IF stagingFunnel.enable THEN
stagingFunnel(
	openingDelay := HMIData.stagingFunnelOpenDelay, 
	openingDwell := HMIData.stagingFunnelOpeningTime,
	closingDwell := HMIData.stagingFunnelClosingTime,
	iOpened := iStagingFunnelOpened, 
	iClosed := iStagingFunnelClosed,  
	oClose => oStagingFunnelCloseOrPerfBreakerDown, 
	oOpen => oStagingFunnelOpenOrPerfBreakerUp
);
END_IF
	 
CASE HMIData.funnelFactorySelection OF
	FunnelSelection.NotInstalled:
		// Disable both funnels
		funnel.enable := FALSE;
		stagingFunnel.enable := FALSE;
		
	FunnelSelection.FunnelWithSensors:
		//
		funnel.enable := HMIData.funnelInUse;
		funnel.feedback := eActuatorFeedbackType.Both;
		stagingFunnel.enable := FALSE;
	
	FunnelSelection.FunnelWithoutSensors:
		//
		funnel.enable := HMIData.funnelInUse;
		funnel.feedback := eActuatorFeedbackType.None;
		stagingFunnel.enable := FALSE;
		
	FunnelSelection.TwoStageFunnelWithSensors:

		_fillerDroppingProductONS(CLK := filler.droppingProduct);
		IF _fillerDroppingProductONS.OSR THEN
			stagingFunnel.Open();
		ELSIF _fillerDroppingProductONS.OSF THEN
			stagingFunnel.Close();
		END_IF

		//
		funnel.enable := HMIData.funnelInUse;
		funnel.feedback := eActuatorFeedbackType.Both;
		stagingFunnel.enable := HMIData.funnelInUse;
		stagingFunnel.feedback := eActuatorFeedbackType.Both;
			 
	FunnelSelection.BagLoadingTray:
		funnel.enable := HMIData.funnelInUse;
		funnel.feedback := eActuatorFeedbackType.Both;
		stagingFunnel.enable := FALSE;
			 
END_CASE

//
sealBarTempSensor(
	busNodeOK := murrIOBusNode.ok,
	ptrTemperatureBytes := ADR(iHeaterBarTempInputs)
);
	 
//
IF sealBarTempSensor.reconfigureIO THEN
	murrIOBusNode.restartBusnodePulse.Trigger();		 
END_IF

//	 
sealBarHeater(
	enable := NOT safePowerFailure.active,
	temperatureSensor := sealBarTempSensor,
	temperatureSetpoint := TO_REAL(HMIData.sealBarTemperatureSetting),
	heaterPulse => 	oHeaterPulse,
	currentTemp => HMIData.sealBarTemperature
);	  

{region "timers"}
// Timers
sealTimer();
bagOpenFingerDelay();
vacuumHoldTimer(PT := TO_TIME(HMIData.vacuumDwell * 1000));
bagOpenCheckDelay();
bagDropTimer(PT := TO_TIME((HMIData.loadPlateDelay * 1000) + (HMIData.bagDropTime * 1000)));
{endregion}
		  
// Setup of HPA and load plate.  Use .Trigger() to run.
HPA.DwellSetting := TO_UINT(HMIData.hpaDwell * 1000);
HPA(Q => oHPAOn);
hpaServiceOnONS(CLK := HMIData.hpaserviceOn);

triggerLPAWhileFeedingONS(CLK := state.sb.releaseFeed = RELEASE_FEED_STATES.MovingJawOutAndFeedingBag);
IF HMIData.lpaDuringBagFeedEnable AND triggerLPAWhileFeedingONS.OSR THEN
	LPA.DwellSetting := TO_DINT(((bagDelivery.remainingLength - HMIData.bagSkirtLength) / TO_REAL(HMIData.bagForwardSpeed)) * 1000.0);
	LPA.Trigger();
END_IF
LPA(Q => oLPAOn);
	 
CASE HMIData.independentBagDeflatorSelection OF
	BagDeflatorSelection.NotInstalled:					// Disable IBD
		 													enableIBDDeflate := FALSE;
															enableIBDEject := FALSE;
	
	BagDeflatorSelection.IBDStandard:	// Enable IBD
															IF HMIData.IBDDeflateDwellTime <> 0 THEN
																enableIBDDeflate := TRUE;
															ELSE
																enableIBDDeflate := FALSE;
															END_IF
															
															IF HMIData.IBDPackageEjectAssistDwellTime <> 0 THEN
																enableIBDEject := TRUE;
															ELSE
																enableIBDEject := FALSE;
															END_IF
	 														
																 
	BagDeflatorSelection.IBDWithHingedPlate:	// Enable IBD with Hinged Plate
															
																 
	BagDeflatorSelection.MotorizedIBD:			// Enable motorized IBD
															IF HMIData.IBDDeflateDwellTime <> 0 THEN
																enableIBDDeflate := TRUE;
															ELSE
																enableIBDDeflate := FALSE;
															END_IF
															
															IF HMIData.IBDPackageEjectAssistDwellTime <> 0 THEN
																enableIBDEject := TRUE;
															ELSE
																enableIBDEject := FALSE;
															END_IF
END_CASE
		
(*  
CASE HMIData.bofSelection OF
	BagOpenFingersSelection.NotInstalled:					// Disable Bag Open
		 													enableBagOpen := FALSE;
															
	
	BagOpenFingersSelection.PneumaticWithBagOpenSensors:	// Enable Bag Open
															enableBagOpen := TRUE;
	
END_CASE
	 *)
		  enableBagOpen := HMIData.bagOpenEnable;

CASE HMIData.cycleStartButtonSelection OF
	PalmButtonSelection.NotInstalled:					// Dont' allow input to start bagger cycle
		 												startCycleReqFromPalmButtons := FALSE;
		 
	PalmButtonSelection.SinglePalmButton:				// Start using one side only
		 												startCycleReqFromPalmButtons := iRightPalmButton;
														
														// Trigger fault if left palm button is seen - should be set up for dual!	 
														IF iLeftPalmButton THEN
															palmButtonConfigError.Trigger();		 
														END_IF
		 
	PalmButtonSelection.DualPalmButton:					// Both buttons must be pressed
		 												startCycleReqFromPalmButtons := iRightPalmButton AND iLeftPalmButton;
															 
	PalmButtonSelection.LightedPalmButton:				
		// Lighted Murr palm button input comes from IO Link
		startCycleReqFromPalmButtons := iMurrTouchButtonOneStatus.0 OR iMurrTouchButtonTwoStatus.0;
		basicLightedPalmButton(
			baggerReady:= readyToRun AND NOT HMIData.sealBarNotAtTemperature.active, 
			baggerFaulted:= HMIData.faultActive, 
			baggerInCycle:= HMIData.inCycle, 
		);
		oMurrTouchbuttonOneState := oMurrTouchButtonTwoState := basicLightedPalmButton.IOLinkStateOutput;													 
														
    PalmButtonSelection.LightedPalmButtonAdvanced, PalmButtonSelection.DualLightedPalmButtonAdvanced:		
		// Lighted Murr palm button input comes from IO Link
		startCycleReqFromPalmButtons := iMurrTouchButtonOneStatus.0 OR iMurrTouchButtonTwoStatus.0;														 
		advancedLightedPalmButtonOne(
			IOLinkData := ADR(oMurrTouchButtonOneIOLinkOutputs),
			baggerReady := readyToRun 
							AND (NOT HMIData.sealBarNotAtTemperature.active) 
							AND (NOT HMIData.stopMachine) ,
			baggerFaulted := HMIData.faultActive,
			baggerInCycle := HMIData.inCycle,
			baggerExternalInhibited := printAndApply.state = PRINT_AND_APPLY_STATES.Inhibited,
			baggerHeatingUp := HMIData.sealBarNotAtTemperature.active AND sealBarHeater.heating,
			baggerCoolingDown := HMIData.sealBarNotAtTemperature.active AND sealBarHeater.cooling AND sealBarHeater.enable
		);	
        IF HMIData.cycleStartButtonSelection = PalmButtonSelection.DualLightedPalmButtonAdvanced THEN
			advancedLightedPalmButtonTwo(
				IOLinkData := ADR(oMurrTouchButtonTwoIOLinkOutputs),
				baggerReady := readyToRun 
							AND (NOT HMIData.sealBarNotAtTemperature.active) 
							AND (NOT HMIData.stopMachine) ,
				baggerFaulted := HMIData.faultActive,
				baggerInCycle := HMIData.inCycle,
				baggerExternalInhibited := printAndApply.state = PRINT_AND_APPLY_STATES.Inhibited,
				baggerHeatingUp := HMIData.sealBarNotAtTemperature.active AND sealBarHeater.heating,
				baggerCoolingDown := HMIData.sealBarNotAtTemperature.active AND sealBarHeater.cooling AND sealBarHeater.enable
			);	
		END_IF					  									 
END_CASE
startCycleReqFromPalmButtonsONS(CLK := startCycleReqFromPalmButtons);	 

// Stack Light active only if no 2nd palm button selected - they use the same IOLink port
IF HMIData.cycleStartButtonSelection <> PalmButtonSelection.DualLightedPalmButtonAdvanced THEN
	stackLight(
		IOLinkData:= ADR(oMurrStackLightOutputs), 
		baggerReady := readyToRun AND NOT HMIData.sealBarNotAtTemperature.active AND NOT HMIData.faultActive ,
		baggerFaulted := HMIData.faultActive,
		baggerInCycle := HMIData.inCycle,
		baggerExternalInhibited := printAndApply.state = PRINT_AND_APPLY_STATES.Inhibited ,
		bagsLow:= HMIData.bagLevelLow.active, 
		bagOpenRetryActive:= bagOpenRetryCount <> 0,
		baggerHeatingUp := HMIData.sealBarNotAtTemperature.active AND sealBarHeater.heating
	);	 
END_IF

		 
_auxIOPhysical(
	state := state,
	configIn1 := iAuxConfigInput1, 
	configIn2 := iAuxConfigInput2,
	bagsLow := HMIData.bagLevelLow.active,
	faultActive := HMIData.faultActive,
	inhibitCycle := printAndApply.inhibitCycle,
	printerDataReady := printerDataReady,
	waitingForFiller := filler.waitingForFiller,
	runExitConveyor := oRunExternalExitConveyor,
	fillerType := HMIData.fillerFactorySelection,
	factorySelection := HMIData.auxIOConfig,
	baggerOK => oAuxBaggerOk,
	readyForFiller => oAuxReadyForFiller,
	inhibitBagger => ,
	configOut1 => oAuxConfigOut1,
	configOut2 => oAuxConfigOut2,
);
	 
		  
_auxIORemote(
	state := state,	
	bagsLow := HMIData.bagLevelLow.active,
	faultActive := HMIData.faultActive,
	inhibitCycle := printAndApply.inhibitCycle,
	printerDataReady := printerDataReady,
	waitingForFiller := filler.waitingForFiller,
	runExitConveyor := oRunExternalExitConveyor,	
	activeFaults := GlobalObjects.CollectionOfActiveFaults.ObjNames,
	inhibitBagger => 
);

HMIData.baggerInhibited.active := _auxIORemote.inhibitBagger  OR _auxIOPhysical.inhibitBagger;

// Filler and EZFeed conveyor setup
CASE HMIData.fillerFactorySelection OF
	FillerSelection.NotInstalled:					// No filler
		// No filler
		 											filler.enable := FALSE;
													filler.activateFiller := FALSE;	
													HMIData.fillerEnable := FALSE;
													ezfeed.enable := FALSE;
													fillerModeCycleStartOnlyPulse.Reset();
													Infeed_Conveyor_IO.Enable := FALSE;
		 
	FillerSelection.StandardFiller:					
													// Only enable filler if Aux IO is enabled
		 											filler.enable := ((HMIData.auxIOConfig.factorySelection = AuxiliaryIOSelection.AuxIOStandard)
																		OR HMIData.auxIOSource.ModbusTCP
																		OR HMIData.auxIOSource.OPC_UA);
													Infeed_Conveyor_IO.Enable := FALSE;
														 
	FillerSelection.EZFeed:							
		filler.enable := TRUE;
		 											ezfeed.enable := TRUE;
													Infeed_Conveyor_IO.Enable := TRUE;
													
END_CASE 	 

ezfeed(
	enable:= , 
	baggerFaulted:= HMIData.faultActive, 
	enableEZFeed:= HMIData.fillerEnable, 
	continuousModeEnable:= HMIData.infeedConveyorRunningMode, 
	partsCountingModeEnable:= HMIData.infeedConveyorCountingMode, 
	flightPresentSensor:= iInfeedFlightSensor, 
	partPresentSensor:= NOT iLightCurtainsClear AND HMIData.lightCurtainSelection = LightCurtainsSelection.LoadingAreaLightCurtains, 
	waitingForFiller:= filler.waitingForFiller AND (NOT HMIData.stopMachine) AND NOT HMIData.batchCountDone.active, 
	indexDwellSetting:= HMIData.infeedIndexDwellTimer, 
	flightTarget:= HMIData.infeedFlightCountTarget, 
	partsTarget:= HMIData.infeedPartsCountTarget, 
	emptyPartsWarningSetting:= HMIData.infeedEmptyPartsSetting, 
	restartFromEmptyParts:= HMIData.initiateCycle, 
	state=> , 
	runVFD=> oRunInfeedVFD, 
	flightCount=> HMIData.infeedFlightCountActual, 
	partsCount=> HMIData.infeedPartsCountActual, 
	emptyPartsWarningCount=> HMIData.infeedEmptyPartsActual, 
	emptyPartsWarning=> HMIData.infeedConveyorOutOfParts.active,
	EZFeedDone=> );

IF HMIData.fillerFactorySelection = FillerSelection.EZFeed THEN
	Infeed_Conveyor_IO.Enable := TRUE; 

	IF Infeed_Conveyor_IO.eState <> IoDrvEthernetIP.AdapterState.RUNNING THEN 
		infeedConveyorIOCommFail.Trigger();
	END_IF
ELSE
	Infeed_Conveyor_IO.Enable := FALSE;
END_IF
	 
infeedConveyorVFDFaulted.faultTrigger := (HMIData.fillerFactorySelection = FillerSelection.EZFeed) AND ezfeed.enableEZFeed AND NOT iInfeedVFDNotFaulted;
		 
fillerModeCycleStartOnlyPulse.DwellSetting := 4000;
fillerModeCycleStartOnlyPulse(Q => HMIData.fillerModeCycleStartOnly.active);
filler(
	enable:= ,	
	inCycle := HMIData.inCycle,
	fillerTrigger:= (iAuxFillerTrigger AND HMIData.auxIOSource.Physical) OR ezfeed.EZFeedDone OR (RemoteComms.OPCInputsToBagger.fillerTrigger AND HMIData.auxIOSource.OPC_UA) OR (RemoteComms.modbusInputsToBagger.fillerTrigger AND HMIData.auxIOSource.ModbusTCP), 
	activateFiller:= HMIData.fillerEnable, 
	dropTime:= HMIData.fillerDropTime,
	state=> , 
	fillerModeActive=> , 
	waitingForFiller=> ,
	cycleBagRequest=> , 
	cycleBaggerToActivateFiller=> , 
	notReady=> 
);
	 
IF filler.activateFiller AND NOT filler.cycleBaggerToActivateFiller.active THEN
	IF HMIData.initiateCycle OR startCycleReqFromPalmButtons THEN
		fillerModeCycleStartOnlyPulse.Trigger();
	END_IF
END_IF

//
loadShelf(
	faultActive := HMIData.faultActive,
	switchedPowerON := iEStopOK,
	inUse := HMIData.loadPlateInUse,
    shakerEnable := HMIData.shakerInstalled,
	shakeStart := HMIData.loadShelfShakerStart,
	shakerDwell := HMIData.loadShelfShakerDwell,
	shakerDelay := HMIData.loadShelfShakerDelay,
	shakerOnDwell := HMIData.loadShelfShakerOnDuration,
	shakerOffDwell := HMIData.loadShelfShakerOffDuration,
	disabledPosition := HMIData.packageEjectDisabledPosition,
	dischargeOnFault := printAndApply.enable,
	faultsEnabled := FALSE,
	moveToLoadingPositon => oLoadShelfUp,
	moveToDischargePosition => oLoadShelfDown
);		 
HMIData.loadShelfService.extendedFeedback := rearLoadPlate.inLoadingPosition;
HMIData.loadShelfService.retractedFeedback := rearLoadPlate.inDischargePosition;

//	 
rearLoadPlate(
	faultActive := HMIData.faultActive,
	switchedPowerON := iEStopOK,
	inUse := HMIData.loadPlateInUse,
	inLoadingPosition := iLoadPlateExtended,
	inDischargePosition := iLoadPlateRetracted,
    shakerEnable := HMIData.shakerInstalled,
	shakeStart := HMIData.rearloadPlateShakerStart,
	shakerDwell := HMIData.rearLoadPlateShakerDwell,
	shakerDelay := HMIData.rearLoadPlateShakerDelay,
	shakerOnDwell := HMIData.rearLoadPlateShakerOnDuration,
	shakerOffDwell := HMIData.rearLoadPlateShakerOffDuration,
	disabledPosition := HMIData.packageEjectDisabledPosition,
	dischargeOnFault := printAndApply.enable,
	moveToLoadingPositon => oloadPlateExtend,
	moveToDischargePosition => oLoadPlateRetract,
	failedToExtend => rearLoadPlateFaults.failedToLoad.faultTrigger,
	failedToRetract => rearLoadPlateFaults.failedToDischarge.faultTrigger
);		 
HMIData.rearLoadPlateService.extendedFeedback := HMIData.loadPlateService.extendedFeedback := rearLoadPlate.inLoadingPosition;
HMIData.rearLoadPlateService.retractedFeedback := HMIData.loadPlateService.retractedFeedback :=  rearLoadPlate.inDischargePosition;

//	 
frontLoadPlate(
	faultActive := HMIData.faultActive,
	switchedPowerON := iEStopOK,
	inUse := HMIData.loadPlateInUse,
	inLoadingPosition := iFrontLoadPlateRetracted,
	inDischargePosition := iFrontLoadPlateExtended,
	//triggerDwell := HMIData.loadPlateDwell,
	//triggerDelay := HMIData.loadPlateDelay,
    shakerEnable := HMIData.shakerInstalled,
	shakeStart := HMIData.frontloadPlateShakerStart,
	shakerDwell := HMIData.frontLoadPlateShakerDwell,
	shakerDelay := HMIData.frontLoadPlateShakerDelay,
	shakerOnDwell := HMIData.frontLoadPlateShakerOnDuration,
	shakerOffDwell := HMIData.frontLoadPlateShakerOffDuration,
	disabledPosition := HMIData.packageEjectDisabledPosition,
	dischargeOnFault := printAndApply.enable,
	moveToLoadingPositon => oFrontLoadPlateToLoad,
	moveToDischargePosition => oFrontLoadPlateToDischarge,
	failedToExtend => forwardLoadPlateFaults.failedToLoad.faultTrigger,
	failedToRetract => forwardLoadPlateFaults.failedToDischarge.faultTrigger
);		 
HMIData.forwardLoadPlateService.extendedFeedback := frontLoadPlate.inLoadingPosition;
HMIData.forwardLoadPlateService.retractedFeedback := frontLoadPlate.inDischargePosition;

CASE HMIData.packageEjectSelection OF
	PackageEjectionSelection.NotInstalled:				// Disable All
		 												loadShelf.enable := FALSE;	
														rearLoadPlate.enable := FALSE;
														frontLoadPlate.enable := FALSE;
														rearLoadPlate.faultsEnabled := FALSE;
														frontLoadPlate.faultsEnabled := FALSE;	
		 
	PackageEjectionSelection.RearRetractingLoadPlate:	// Enable Rear Retracting Load Plate
		 												loadShelf.enable := FALSE;	
														rearLoadPlate.enable := TRUE;
														frontLoadPlate.enable := FALSE;
														rearLoadPlate.faultsEnabled := powerSettlingTimer.Q;
														frontLoadPlate.faultsEnabled := FALSE;			
														rearLoadPlate.triggerDelay := HMIData.loadPlateDelay;
														rearLoadPlate.triggerDwell := HMIData.loadPlateDwell;
	
	PackageEjectionSelection.LabelSideUp:				// Enable All
		 												loadShelf.enable := TRUE;	
														rearLoadPlate.enable := TRUE;
														frontLoadPlate.enable := TRUE;
														rearLoadPlate.faultsEnabled := powerSettlingTimer.Q;
														frontLoadPlate.faultsEnabled := state.head >= HEAD_STATES.ReleaseAndFeedBag;
                                                        rearLoadPlate.triggerDelay := HMIData.loadPlateDelay;
														rearLoadPlate.triggerDwell := HMIData.loadPlateDwell + HMIData.loadPlateDelay;
														loadShelf.triggerDelay := HMIData.loadShelfDelay;
														loadShelf.triggerDwell := HMIData.loadShelfDwell;
														frontLoadPlate.triggerDelay := HMIData.loadShelfDelay;
														frontLoadPlate.triggerDwell := HMIData.loadShelfDwell;
															 
	PackageEjectionSelection.RearRetractWithRetractShelf:   
														// Enable Rear Retracting Load Plate and Shelf
		 												loadShelf.enable := TRUE;	
														rearLoadPlate.enable := TRUE;
														frontLoadPlate.enable := FALSE;
														rearLoadPlate.faultsEnabled := powerSettlingTimer.Q;
														frontLoadPlate.faultsEnabled := FALSE;
														rearLoadPlate.triggerDelay := HMIData.loadPlateDelay;
														rearLoadPlate.triggerDwell := HMIData.loadPlateDwell;
														loadShelf.triggerDelay := HMIData.loadShelfDelay;
														loadShelf.triggerDwell := HMIData.loadShelfDwell;
END_CASE	
	 

//  
exitConveyorRun();
exitConveyorRun.DwellSetting := TO_DINT(HMIData.exitConveyorDwell * 1000);
exitConveyorJogONS(CLK := HMIData.exitConveyorJog);

oRunExitConveyor := ((exitConveyorRun.Q OR collisionDetection.runExitConveyor OR (printAndApply.runConveyorAfterApply AND NOT printAndApply.inhibitConveyor)) AND HMIData.integratedExitConveyorSelection = IntegratedConveyorSelection.RearExit);
	 
_runIntegratedExitConveyor := ((exitConveyorRun.Q OR collisionDetection.runExitConveyor OR (printAndApply.runConveyorAfterApply AND NOT printAndApply.inhibitConveyor)) AND HMIData.integratedExitConveyorSelection = IntegratedConveyorSelection.RearExit);	 
oRunExitConveyorForward := _runIntegratedExitConveyor AND NOT (HMIData.reverseConveyor OR _auxIOPhysical.reverseConveyor OR _auxIORemote.reverseConveyor);
oRunExitConveyor := oRunExitConveyorForward;
oRunExitConveyorReverse := _runIntegratedExitConveyor AND (HMIData.reverseConveyor OR _auxIOPhysical.reverseConveyor OR _auxIORemote.reverseConveyor);
	 //Aux IO conveyore control
oAuxExitConveyorForward := _runIntegratedExitConveyor; 
oAuxExitConveyorReverse := HMIData.reverseConveyor OR _auxIOPhysical.reverseConveyor OR _auxIORemote.reverseConveyor;


 
externalExitConveyorRun();
externalExitConveyorRun.DwellSetting := TO_UINT(HMIData.externalExitConveyorDwell * 1000);
externalExitConveyorJogONS(CLK := HMIData.externalExitConveyorJog);

oRunExternalExitConveyor := collisionDetection.runExternalExitConveyor 
							OR externalExitConveyorRun.Q
							OR (printAndApply.runConveyorAfterApply  
								AND NOT collisionDetection.inhibitExternalExitConveyor 
								AND HMIData.externalExitConveyorSelection <> ExteralConveyorSelection.NotInstalled) 
							AND NOT barcodeVerificationFailed.active;
//oRunExternalExitConveyor := collisionDetection.runExternalExitConveyor OR externalExitConveyorRun.Q OR printAndApply.runConveyorAfterApply AND NOT collisionDetection.inhibitExternalExitConveyor AND HMIData.externalExitConveyorSelection <> ExteralConveyorSelection.NotInstalled;	  
	  
IF printAndApply.inhibitConveyor THEN
	exitConveyorRun.ManualOFf();
	externalExitConveyorRun.ManualOFf();
END_IF	 
		  
bagOpenFingers(enable := HMIData.bofSelection <> BagOpenFingersSelection.NotInstalled,
				releaseOutput => oBOFUp,
		 		grabOutput => oBOFDown,
				rightFingerBagPresent := iRightFingerBagPresent,
				leftFingerBagPreset := iLeftFingerBagPresent,
				bagFailedToGrabBothFingersCount := Globals.bagFailedToGrabBothFingersCount,
				bagFailedToGrabLeftFingerCount := Globals.bagFailedToGrabLeftFingerCount,
				bagFailedToGrabRightFingerCount := Globals.bagFailedToGrabRightFingerCount,
				successfulBagOpenCount := Globals.successfulBagOpenCount);

// Setup and run adjustable passthrough
//refIECObject := Pbar_ServoEIP;

IBD_Motor.Enable := HMIData.independentBagDeflatorSelection = BagDeflatorSelection.MotorizedIBD;	 
IBDMotor(ptrEIPInputs := ADR(iIBDMotorEIP),
                ptrEIPOutputs := ADR(oIBDMotorEIP),
                stepsPerInchSetpoint := Globals.STEPS_PER_INCH_TFBelt,
				reversePolarity := FALSE,
				defaultCurrentSetpoint := 650,
				commFail := IBD_Motor.eState <> IoDrvEthernetIP.AdapterState.RUNNING AND IBD_Motor.Enable,
				isHomable := TRUE);
IBDMotor.Execute();

// Clamp maximim IBD open position - 9" for Pro 18, 12" for Pro 24
IF HMIData.passthroughSetting + HMIData.IBDOffset > Globals.maximumPassthough THEN
	 IBDOutSetting := Globals.maximumPassthough;
ELSE
	IBDOutSetting := HMIData.passthroughSetting + HMIData.IBDOffset;
END_IF
		  
IBD(
	enable:= , 
	pbarOutSetting:= IBDOutSetting, 
	inPositionSetting:= HMIData.IBDClosePosition, 
	disableFaults:= , 
	extendCommand:= HMIData.IBDService.extendCommand, 
	retractCommand:= HMIData.IBDService.retractCommand ,  
	failToOpen=> , 
	state=> , 
	actualPosition=> , 
	IBDOpen=> , 
	homeRequired=> , 
	clamped=> , 
	IBDMotor:= IBDMotor,
	failedToHome=> );
IBDFailedToHome.faultTrigger := IBD.failedToHome AND (HMIData.independentBagDeflatorSelection = BagDeflatorSelection.MotorizedIBD);
	 
obstructionFaultONS(CLK := (pressureBar.faults.obstructionDetected.active OR pressureBar.faults.failedToClose.active));
IF obstructionFaultONS.OSR THEN
	IBD.RemovePower();
END_IF
		 
IF HMIData.IBDService.extendCommand THEN
	HMIData.IBDService.extendCommand := FALSE;
END_IF
	 
IF HMIData.IBDService.retractCommand THEN
	HMIData.IBDService.retractCommand := FALSE;
END_IF
{endregion}
	 
hmiLight(lightOutput => oHMILight);
faultONS(CLK := HMIData.faultActive);

readyToRun := (motorizedSealFlatteners.Ready OR NOT motorizedSealFlatteners.enable) 
                AND (pressureBar.Ready OR NOT pressureBar.enable)
				AND (IBD.Ready OR NOT enableIBDDeflate)
                AND (bagDelivery.Ready OR NOT bagDelivery.enable)
                AND (zebraPrinter.Ready OR NOT zebraPrinter.enable)
				AND (NOT oSealBarExtend)
				AND murrIOBusNode.ok;	

iPowerOffButtonONS(CLK := iPowerOffButton);
resetTimer(IN := iPowerOffButtonONS.OSR);

allMotorCommsGood := NOT motorizedSealFlatteners.sealFlattenersHorizontalAxisMotor.faults.commFail.active
					AND NOT IBDMotor.faults.commFail.active
					AND NOT pressureBarMotor.faults.commFail.active
					AND NOT bagDelivery.bagFeedMasterMotor.faults.commFail.active
					AND NOT bagDelivery.bagFeedRearMotor.faults.commFail.active;

IF iPowerOffButtonONS.OSR THEN
	reset();
END_IF
			
IF HMIData.makeReady OR resetTimer.Q THEN
	posInhibit := pressureBar.jawClear OR pbarSensorBypass;
	Cube67_BN_E_V2.xAcknowledge := TRUE;
	FestoManifold.xAcknowledge := TRUE;
	MSFMotor.xAcknowledge := TRUE;
	Bag_Delivery_EIP_Motor.xAcknowledge := TRUE;
	Pbar_ServoEIP.xAcknowledge := TRUE;
	Bag_Delivery_Rear_Motor.xAcknowledge := TRUE;
	Keyence_BCV.xAcknowledge := TRUE;
	IBD_MOtor.xAcknowledge := TRUE;
	Panther_PA.xAcknowledge := TRUE;
	
	HMIData.ackAllFaults := TRUE;
	enable := TRUE;
	
	printAndApply.Reset();
	
	bagDropTimer.IN := FALSE;
	
	motorizedSealFlattenersMode := DEVICE_MODES.Auto;
	motorizedSealFlatteners.Reset();
	
	HMIData.bagOpenFeedNewBagCount := 0;
	bagOpenRetryCount := 0;
	
	HMIData.stopMachine := FALSE;
	HMIData.inCycle := FALSE;
	electricPressureBarMode := DEVICE_MODES.Auto;
	
	pressureBar.enable := TRUE;
	enableHeater := TRUE;
	
	bagDeliveryMode := DEVICE_MODES.Auto;
	bagDelivery.Reset();
	bagDelivery.enable := TRUE;
	
	IF NOT bagOpenFingers.CheckIfBagGrabbed(FALSE) THEN
		bagOpened := FALSE;
	END_IF

	printerMode := DEVICE_MODES.Auto;
	zebraPrinter.Reset();
	
	IF iPowerOffButtonONS.OSR AND NOT bagDelivery.bagTensionFault.active THEN
		IF (HMIData.factoryTestMode AND (HMIData.bagsMade.count < 1000)) THEN
			HMIData.bagsMade.Clear();
		END_IF 
	END_IF  
	
	pressureBarMotor.Reset();
	passthroughMode := DEVICE_MODES.Auto;

	oVacOn := FALSE;
	rearLoadPlate.Reset();
	frontLoadPlate.Reset();
	loadShelf.Reset();
	collisionDetection.Reset();
	
	LPA.Reset();
	LPA.ManualOff();
	HPA.Reset();
	IF (HMIData.funnelFactorySelection = FunnelSelection.BagLoadingTray) THEN
		IF pressureBar.pressureBarOpen THEN
			funnel.Open();
		ELSE
			funnel.Close();
		END_IF
	ELSE
		funnel.Close();
	END_IF
	
	exitConveyorRun.Reset();
	externalExitConveyorRun.Reset();
	oSealBarExtend := FALSE;
	oSealBarRetract := TRUE;
	sealTimer.IN := FALSE;
	pressureBarCloseDelay.IN := FALSE;
	filler.Reset();
	_auxIOPhysical.Reset();
	fillerModeCycleStartOnlyPulse.Reset();
	barcodeVerifier.Reset();
	keyenceBCV.Reset();
	state.head := HEAD_STATES.Idle;
	setPassthroughPB := FALSE;
	HMIData.jobLoadRequired.active := TRUE;
	HMIData.makeReady := FALSE;
	hmiLight.TurnOff();
	autoModeKeepCycling := FALSE;
	
ELSE
	Cube67_BN_E_V2.xAcknowledge := FALSE;
	FestoManifold.xAcknowledge := FALSE;
	MSFMotor.xAcknowledge := FALSE;
	Bag_Delivery_EIP_Motor.xAcknowledge := FALSE;
	Pbar_ServoEIP.xAcknowledge := FALSE;
	Bag_Delivery_Rear_Motor.xAcknowledge := FALSE;
	Keyence_BCV.xAcknowledge := FALSE;
	IBD_MOtor.xAcknowledge := FALSE;
	Panther_PA.xAcknowledge := FALSE;
END_IF

IF enableONS.Q OR resetONS.Q THEN
    state.head := HEAD_STATES.Idle;
	state.sb.sealSeparate := SEAL_SEPARATE_STATES.Idle;
	state.sb.releaseFeed := RELEASE_FEED_STATES.Idle;
	state.sb.openBag := BAG_OPEN_ASSIST_STATES.Idle;
	state.sb.finishCycle := FINISH_CYCLE_STATES.Idle;
	state.sb.automation := AUTOMATION_STATES.Idle;
	state.sb.printOutOfCycle := PRINT_OUT_OF_CYCLE_STATES.Idle;
	motorizedSealFlatteners.Reset();
	pressureBar.Reset();
	IBD.Reset();
	bagDelivery.bagFeedRearMotor.EnableTensionFault();
	bagDelivery.AutoFeedToEye();
// 	bagDelivery.Reset();
	zebraPrinter.Reset();
	homeJawPB := FALSE;

	IF IBD.homeRequired THEN
		homeJawPB := TRUE;
	ELSE
		homeJawPB := TRUE;
	END_IF
	IF pressureBar.homeRequired THEN
		homeJawPB := TRUE;
	ELSE
		homeJawPB := TRUE;
	END_IF

	bagDropTimer.IN := FALSE;
	_reset := FALSE;
	cycleTimer.IN := FALSE;
	
	
	IF NOT (HMIData.mailerMaterial = MAILER_MATERIAL.paper) 
		AND (HMIData.sealAreaOptionSelection = SealAreaOptionSelectionEnum.SealFlattenersWithPerfBreaker) 
		AND NOT stagingFunnel.enable
		THEN				
			oStagingFunnelCloseOrPerfBreakerDown 	:= FALSE;
			oStagingFunnelOpenOrPerfBreakerUp   	:= TRUE;
		END_IF
END_IF

IF HMIData.bagsMade.count >= 1000 THEN
	Globals.factoryTestComplete := TRUE;
END_IF

IF Globals.factoryTestComplete THEN
	HMIData.machineNotTested.active := FALSE;
ELSE
	HMIData.machineNotTested.active := TRUE;
END_IF

IF HMIData.factoryTestMode THEN
	HMIData.factoryTestModeActive.active := TRUE;
ELSE
	HMIData.factoryTestModeActive.active := FALSE;
END_IF

// Disable the printer on dry cycle because we dont't want to print on the platen roller               
IF HMIData.enableDryCycle THEN
    zebraPrinter.enable := FALSE;
END_IF

// Send torque value to motor                 
rearMotorCommsReturned(CLK := bagDelivery.bagFeedRearMotor.commFail);
IF HMIData.jobLoaded OR rearMotorCommsReturned.Q THEN
	bagDelivery.bagFeedRearMotor.SetTorque((TO_DINT(HMIData.bagTensionSetting * 100)));
END_IF

// Clear batch count on batch enable
batchEnableONS(CLK := HMIData.batchEnable);
IF (batchEnableONS.OSR)
	OR (NOT HMIData.batchEnable) 
	OR (HMIData.batchReset)
	OR (resetONS.Q AND HMIData.batchCountDone.active)
THEN
    HMIData.batchCount := 0;
	HMIData.batchReset := FALSE;
END_IF
HMIData.batchCountDone.active := (HMIData.batchCount >= HMIData.batchSetting) AND HMIData.batchEnable;
IF HMIData.batchCountDone.active OR NOT HMIData.autoEnable OR HMIData.fillerEnable THEN
	autoModeKeepCycling := FALSE;
END_IF

//IF NOT enable OR NOT readyToRun OR faultONS.OSR THEN
IF NOT enable OR faultONS.OSR THEN
	state.head := HEAD_STATES.Fault;
	//pressureBarMotor.Stop();
	cycleTimer.IN := FALSE;
END_IF
pressureBarCloseDelay(PT := TO_TIME(HMIData.pressureBarCloseDelay * 1000));
cycleTimer();
autoModeKeepCyclingTimer(PT := TO_TIME(HMIData.autoModeDwell * 1000), IN := autoModeKeepCycling AND state.head = HEAD_STATES.Idle);

HMIData.mayCycleUnexpectedly.active := autoModeSelected OR filler.activateFiller;

footSwitchONS(CLK := iFootSwitch);
_bagGrabbedONS(CLK := _auxIOPhysical.bagGrabbed OR _auxIORemote.bagGrabbed);

IF state.head <> HEAD_STATES.Idle AND HMIData.initiateCycle THEN
	HMIData.initiateCycle := FALSE;
END_IF
CASE state.head OF
    HEAD_STATES.Idle :                              // Start cycle if enabled
                                                    IF (startCycle AND (filler.cycleBaggerToActivateFiller.active OR NOT filler.activateFiller)
													OR (HMIData.factoryTestMode AND (HMIData.bagsMade.count < 1000)) AND (factoryTestModeKeepCycling AND NOT LPA.Q)
													OR (startCycleReqFromPalmButtonsONS.OSR) AND (filler.cycleBaggerToActivateFiller.active OR NOT filler.activateFiller)
													OR (HMIData.initiateCycle) AND (filler.cycleBaggerToActivateFiller.active OR NOT filler.activateFiller)
													OR (filler.cycleBagRequest AND HMIData.autoEnable)
													OR (filler.cycleBagRequest AND NOT HMIData.autoEnable) AND (footSwitchONS.OSR OR HMIData.initiateCycle OR startCycleReqFromPalmButtonsONS.OSR)
													OR (autoModeKeepCyclingTimer.Q)
													OR footSwitchONS.OSR AND (filler.cycleBaggerToActivateFiller.active OR NOT filler.activateFiller))
													AND (NOT HMIData.sealBarNotAtTemperature.active OR HMIData.enableDryCycle)
													AND NOT barcodeVerificationFailed.active
													AND NOT HMIData.faultActive 
													AND NOT HMIData.stopMachine 
													AND NOT HMIData.baggerInhibited.active
													AND NOT HMIData.batchCountDone.active
													AND NOT setPassthroughPB
													AND NOT printAndApply.clearOutBaggerIndicaiton
													AND readyToRun 
													THEN
														posInhibit := TRUE;
                                                        startCycle := FALSE;
														cycleTimer.IN := TRUE;
														HMIData.initiateCycle := FALSE;
														state.head := HEAD_STATES.SealAndSeparateBag;
														IF bagOpenFingers.CheckIfBagGrabbed(FALSE) THEN
															bagOpened := TRUE;
														END_IF
                                                    END_IF
													
													IF HMIData.baggerProfileSelection = BaggerProfile.EQ22085 THEN
														IF _bagGrabbedONS.Q THEN
															state.head := HEAD_STATES.PrepareForAutomatedBagRemoval;
														END_IF
                                                    END_IF
													IF NOT Globals.passthroughChangedFromJog AND HMIData.jobLoaded THEN
														HMIData.jobLoaded := FALSE;
													END_IF
                                                    IF (TO_DINT(HMIData.passthroughSetting*1000) <> TO_DINT(passthroughSettingLast*1000)) OR (Globals.passthroughChangedFromJog AND HMIData.jobLoaded) AND NOT pressureBarMotor.Faulted AND NOT pressureBarMotor.HomeRequired THEN
															setPassthroughPB := TRUE;
															Globals.passthroughChangedFromJog := FALSE;
															HMIData.jobLoaded := FALSE;
															passthroughSetting := HMIData.passthroughSetting;
															passthroughSettingLast := HMIData.passthroughSetting;
													END_IF
													
													IF (NOT (pressureBarMotor.HomeRequired OR pressureBarMotor.Faulted))
														AND ((NOT motorizedSealFlatteners.sealFlattenersHorizontalAxisMotor.homeRequiredIndication OR motorizedSealFlatteners.sealFlattenersHorizontalAxisMotor.Faulted) OR NOT motorizedSealFlatteners.enable)
														AND readyToRun 
														AND NOT HMIData.faultActive
													THEN
														hmiLight.TurnOn();
													END_IF
													
													IF HMIData.stopMachine THEN
														setPassthroughPB := FALSE;
														homeJawPB := FALSE;
														startCycle := FALSE;
														HMIData.initiateCycle := FALSE;
														factoryTestModeKeepCycling := FALSE;
														autoModeKeepCycling := FALSE;
														hmiLight.TurnOff();
														filler.Reset();
														ezFeed.Reset();
														LPA.Reset();
													END_IF
													
													IF HMIData.sealBarNotAtTemperature.active THEN
														factoryTestModeKeepCycling := FALSE;
														autoModeKeepCycling := FALSE;
													END_IF
													
													IF bagOpened THEN
                                                        IF NOT bagOpenFingers.CheckIfBagGrabbed(FALSE) AND NOT HMIData.enableDryCycle THEN
															openedBagWasRemoved.Trigger();
															bagOpened := FALSE;
														END_IF
													END_IF
													posInhibitTON(IN:= posInhibit AND NOT pressureBar.jawClear, PT:= T#500MS);
													IF posInhibitTON.Q THEN
														posInhibit:= FALSE;
													END_IF
													{region:'Service'}
													IF setPassthroughPB AND NOT homeJawPB THEN
														hmiLight.BlinkSlow();
														IF HMIData.passthroughPosition < HMIData.passthroughSetting THEN
															motorizedSealFlatteners.sealFlattenersHorizontalAxisMotor.MoveToPositionTorque(2,1000,1000,2000,125);
														END_IF
														state.head := HEAD_STATES.MovePassthrough;
													END_IF
														
													IF homeJawPB THEN
														hmiLight.BlinkSlow();
														state.head := HEAD_STATES.PassthroughPreCheck;												
													END_IF    
													
													IF HMIData.loadPlateService.retractCommand OR HMIData.rearLoadPlateService.retractCommand THEN
														rearLoadPlate.moveToDischargePos();
														HMIData.loadPlateService.retractCommand := FALSE;
														HMIData.rearLoadPlateService.retractCommand := FALSE;
													END_IF                                      
                                                    
													IF HMIData.loadPlateService.extendCommand OR HMIData.rearLoadPlateService.extendCommand THEN
														rearLoadPlate.moveToLoadingPos();
														HMIData.loadPlateService.extendCommand := FALSE;
														HMIData.rearLoadPlateService.extendCommand := FALSE;
													END_IF
														 
													IF HMIData.perfBreakerService.exhaustCommand  AND HMIData.sealAreaOptionSelection = (SealAreaOptionSelectionEnum.SealFlattenersWithPerfBreaker OR SealAreaOptionSelectionEnum.PerfBreaker)  THEN
														perfBreaker.Exhaust();
														posInhibit:= TRUE;
														HMIData.perfBreakerService.exhaustCommand := FALSE;
													END_IF
													IF HMIData.perfBreakerService.retractCommand  AND HMIData.sealAreaOptionSelection = (SealAreaOptionSelectionEnum.SealFlattenersWithPerfBreaker OR SealAreaOptionSelectionEnum.PerfBreaker) THEN
														perfBreaker.MoveUp();
														posInhibit:= TRUE;
														HMIData.perfBreakerService.retractCommand := FALSE;
													END_IF
													IF HMIData.perfBreakerService.extendCommand  AND HMIData.sealAreaOptionSelection = (SealAreaOptionSelectionEnum.SealFlattenersWithPerfBreaker OR SealAreaOptionSelectionEnum.PerfBreaker) THEN
														perfBreaker.MoveDown();
														posInhibit:= TRUE;
														HMIData.perfBreakerService.extendCommand := FALSE;
													END_IF
													
													IF HMIData.loadShelfService.retractCommand THEN
														loadShelf.moveToDischargePos();
														HMIData.loadShelfService.retractCommand := FALSE;
													END_IF                                      
                                                    
													IF HMIData.loadShelfService.extendCommand THEN
														loadShelf.moveToLoadingPos();
														HMIData.loadShelfService.extendCommand := FALSE;
													END_IF	

													IF HMIData.forwardLoadPlateService.retractCommand THEN
														frontLoadPlate.moveToDischargePos();
														HMIData.forwardLoadPlateService.retractCommand := FALSE;
													END_IF                                      
                                                    
													IF HMIData.forwardLoadPlateService.extendCommand THEN
														frontLoadPlate.moveToLoadingPos();
														HMIData.forwardLoadPlateService.extendCommand := FALSE;
													END_IF	 
													
													IF HMIData.IBDService.retractCommand THEN
														IBD.CloseIBD();
														HMIData.IBDService.retractCommand := FALSE;
													END_IF                                      
                                                    
													IF HMIData.IBDService.extendCommand THEN
														IBD.OpenIBD();
														HMIData.IBDService.extendCommand := FALSE;
													END_IF	
														 
													IF HMIData.funnelService.retractCommand THEN
														funnel.Open();
														HMIData.funnelService.retractCommand := FALSE;
													END_IF                                      
                                                    
													IF HMIData.funnelService.extendCommand THEN
														funnel.Close();
														HMIData.funnelService.extendCommand := FALSE;
													END_IF	
	 													
													IF HMIData.pressureBarService.extendCommand THEN
														pressureBar.OpenJaw();
														HMIData.pressureBarService.extendCommand := FALSE;
													END_IF	
														 
													IF HMIData.pressureBarService.retractCommand THEN
														pressureBar.CloseJaw();
														HMIData.pressureBarService.retractCommand := FALSE;
													END_IF	
														 
													IF HMIData.lpaServicePulse THEN
														LPA.DwellSetting := TO_DINT(HMIData.lpaDwell * 1000);
														LPA.Trigger();
														HMIData.lpaServicePulse := FALSE;
													ELSIF HMIData.lpaServiceOn THEN
														LPA.ManualOn();
														HMIData.lpaServiceOn := FALSE;
													ELSIF HMIData.lpaServiceOff THEN
														LPA.ManualOff();
														HMIData.lpaServiceOff := FALSE;
													END_IF
													
													IF HMIData.vacuumServiceOn THEN
														oVacOn := TRUE;
														HMIData.vacuumServiceOn := FALSE;
													ELSIF HMIData.vacuumServiceOff THEN
														oVacOn := FALSE;
														HMIData.vacuumServiceOff := FALSE;
													END_IF
														 		  
													IF HMIData.hpaServicePulse THEN
														hpa.Trigger();
														HMIData.hpaServicePulse := FALSE;
													ELSIF hpaServiceOnONS.OSR THEN
														HPA.ManualOn();
													ELSIF hpaServiceOnONS.OSF THEN
														HPA.ManualOff();
													END_IF
													
													IF HMIData.exitConveyorStartDwell THEN
														exitConveyorRun.Trigger();
														HMIData.exitConveyorStartDwell := FALSE;
													ELSIF HMIData.exitConveyorStart OR exitConveyorJogONS.OSR THEN
														exitConveyorRun.ManualOn();
														HMIData.exitConveyorStart := FALSE;
													ELSIF HMIData.exitConveyorStop OR exitConveyorJogONS.OSF THEN
														exitConveyorRun.ManualOff();
														HMIData.exitConveyorStop := FALSE;
													END_IF
													
													IF HMIData.externalExitConveyorStartDwell THEN
														externalExitConveyorRun.Trigger();
														HMIData.externalExitConveyorStartDwell := FALSE;
													ELSIF HMIData.externalExitConveyorStart OR externalExitConveyorJogONS.OSR THEN
														externalExitConveyorRun.ManualOn();
														HMIData.externalExitConveyorStart := FALSE;
													ELSIF HMIData.externalExitConveyorStop OR externalExitConveyorJogONS.OSF THEN
														externalExitConveyorRun.ManualOff();
														HMIData.externalExitConveyorStop := FALSE;
													END_IF
	 
													IF HMIData.sealBarServiceCycle THEN
														sealTimer.PT := TO_TIME(HMIData.sealBarDwell * 1000);
														sealTimer.IN := TRUE;
														IF NOT sealTimer.Q THEN
															oSealBarExtend := TRUE;
															oSealBarRetract := FALSE;
														ELSE 
															sealTimer.IN := FALSE;
															oSealBarExtend := FALSE;
															oSealBarRetract := TRUE;
															HMIData.sealBarCycles.Increment();
															HMIData.sealBarServiceCycle := FALSE;
														END_IF
													ELSIF HMIData.sealBarServiceExtend THEN
														oSealBarExtend := TRUE;
														oSealBarRetract := FALSE;
														HMIData.sealBarServiceExtend := FALSE;
													ELSIF HMIData.sealBarServiceRetract THEN
														oSealBarExtend := FALSE;
														oSealBarRetract := TRUE;
														HMIData.sealBarServiceRetract := FALSE;
													END_IF
														 
													IF HMIData.bagOpenFingersServiceGrab THEN
														bagOpenFingers.Grab();
														HMIData.bagOpenFingersServiceGrab := FALSE;
													ELSIF HMIData.bagOpenFingersServiceRelease THEN
														bagOpenFingers.Release();
														HMIData.bagOpenFingersServiceRelease := FALSE;
													END_IF
													{endregion:'Service'}
                                                    
													                                                         
                                                    // Fault if labels stack up in queue 
                                                    IF (printerDataReady AND HMIData.labelsQueuedUpFaultEnable) THEN
                                                        labelsQueuedUpFault.faultTrigger := TRUE;    
                                                    ELSE
                                                        labelsQueuedUpFault.faultTrigger := FALSE;
                                                    END_IF              
														 
    HEAD_STATES.SealAndSeparateBag :                // Begin Seal and Separate State machine
		// Begin Seal and Separate State machine
													IF printAndApply.enable AND bagOpened THEN
														printAndApply.BeginCycle();
													END_IF
													filler.BaggerCycleInitiated();
                                                    HMIData.inCycle := TRUE;
													HMIData.airFilterClean.Increment();
													HMIData.baggerCycles.Increment();
													IF funnel.enable THEN
														funnel.Close();
													END_IF
													
        											state.head := HEAD_STATES.SealingAndSeparatingBag;
													state.sb.sealSeparate := SEAL_SEPARATE_STATES.Shake;
                                                    
    HEAD_STATES.SealingAndSeparatingBag :            IF state.sb.sealSeparate = SEAL_SEPARATE_STATES.Done THEN
                                                        state.head := HEAD_STATES.SealedAndSeparatedBag;
                                                        state.sb.sealSeparate := SEAL_SEPARATE_STATES.Idle;
                                                    END_IF    

    HEAD_STATES.SealedAndSeparatedBag :             state.head := HEAD_STATES.ReleaseAndFeedBag;                                    
                                                    
    HEAD_STATES.ReleaseAndFeedBag :                    // Open the jaw and release the bag
                                                    state.sb.releaseFeed := RELEASE_FEED_STATES.WaitForPressureBarOpenTimer;
                                                    state.head := HEAD_STATES.ReleasingAndFeedingBag;
                                                    
    HEAD_STATES.ReleasingAndFeedingBag :            // 
                                                    IF state.sb.releaseFeed = RELEASE_FEED_STATES.Done THEN
                                                       state.head := HEAD_STATES.ReleasedAndFedBag;
                                                       state.sb.releaseFeed := RELEASE_FEED_STATES.Idle;
                                                    END_IF
                                                    
    HEAD_STATES.ReleasedAndFedBag :                    // 
                                                    {warning 'TODO: change this counting logic to account for MSF'}
                                                    IF HMIData.batchEnable THEN
                                                        HMIData.batchCount := HMIData.batchCount + 1;
                                                    END_IF
  
                                                    IF HMIData.enableDryCycle THEN
                                                        Globals.dryCycleCount := Globals.dryCycleCount + 1;     
                                                    ELSE
                                                        Globals.bagsMadeCount := Globals.bagsMadeCount + 1; 
                                                    END_IF
													IF enableBagOpen THEN
                                                    	state.head := HEAD_STATES.OpenBag;
                                                    ELSE
                                                        state.head := HEAD_STATES.FinishCycle;
                                                    END_IF
                                                                   
    HEAD_STATES.OpenBag :                            // Close jaw to grab the bag
                                                    state.sb.openBag := BAG_OPEN_ASSIST_STATES.MoveJawIn;
                                                    state.head := HEAD_STATES.OpeningBag;
                                                    
                                                    
    HEAD_STATES.OpeningBag :                        // Open jaw and grab onto the bag
                                                    IF state.sb.openBag = BAG_OPEN_ASSIST_STATES.Done THEN
                                                        state.head := HEAD_STATES.OpenedBag;
                                                        state.sb.openBag := BAG_OPEN_ASSIST_STATES.Idle;
													ELSIF state.sb.openBag = BAG_OPEN_ASSIST_STATES.FeedNewBag THEN
														state.head := HEAD_STATES.SealAndSeparateBag;
														state.sb.openBag := BAG_OPEN_ASSIST_STATES.Idle;
                                                    END_IF
                                                    
    HEAD_STATES.OpenedBag :                            // Move fingers in and to bag holding and reset cycle
                                                    IF ((motorizedSealFlatteners.state = SEAL_FLATTENER_STATES.Idle)
														OR (motorizedSealFlatteners.state = SEAL_FLATTENER_STATES.MovedFlattenersIn AND HMIData.funnelFactorySelection = FunnelSelection.BagLoadingTray)	
														OR NOT motorizedSealFlatteners.enable)
														THEN
														state.head := HEAD_STATES.FinishCycle;
                                                    END_IF
	HEAD_STATES.FinishCycle :			//
													state.sb.finishCycle := FINISH_CYCLE_STATES.Start;
													state.head := HEAD_STATES.FinishingCycle;
	HEAD_STATES.FinishingCycle : 		//
													IF state.sb.finishCycle = FINISH_CYCLE_STATES.Done THEN
														state.head := HEAD_STATES.FinishedCycle;
														state.sb.finishCycle := FINISH_CYCLE_STATES.Idle;
													END_IF
	HEAD_STATES.FinishedCycle :			//
											HMIData.bagsMade.Increment();
											HMIData.resettableBagsMade.Increment();
                                            state.head := HEAD_STATES.Idle;
											filler.BaggerCycledAndReady();
											cycleTime := (TIME_TO_REAL(cycleTimer.ET) / 1000); 
											cycleTimer.IN := FALSE;
											IF HMIData.averageCycleTime = 0 THEN
												HMIData.averageCycleTime := cycleTime;
											ELSE
												HMIData.averageCycleTime := (cycleTime + HMIData.averageCycleTime) / 2;
											END_IF
											HMIData.inCycle := FALSE;
											
											IF HMIData.autoEnable AND NOT HMIData.stopMachine AND NOT HMIData.fillerEnable THEN
												autoModeKeepCycling := TRUE;
											END_IF								
											
											IF HMIData.factoryTestMode AND NOT HMIData.stopMachine THEN
												IF (HMIData.bagsMade.count >= 1000) THEN
													factoryTestModeKeepCycling := FALSE;
													HMIData.factoryTestMode := FALSE;
												ELSE
													factoryTestModeKeepCycling := TRUE;
												END_IF
											END_IF	

HEAD_STATES.PassthroughPreCheck :
										IF HMIData.sealAreaOptionSelection = (SealAreaOptionSelectionEnum.SealFlattenersWithPerfBreaker OR SealAreaOptionSelectionEnum.PerfBreaker) THEN
											posInhibit := TRUE;
											IF NOT pressureBar.jawClear AND HMIData.sealAreaOptionSelection = (SealAreaOptionSelectionEnum.SealFlattenersWithPerfBreaker OR SealAreaOptionSelectionEnum.PerfBreaker) THEN
												pressureBar.MoveJawClear();

											END_IF
											IF pressureBar.jawClear THEN
													//waitPassthroughMove:= FALSE;
													state.head := HEAD_STATES.StartHoming;																				
 											END_IF
										ELSE
											state.head := HEAD_STATES.StartHoming;
										END_IF	
		
    HEAD_STATES.StartHoming :            // 
											IF allMotorCommsGood THEN
												motorizedSealFlatteners.sealFlattenersHorizontalAxisMotor.faults.notHomed.Ack();
												IF pressureBar.homeRequired THEN
													pressureBar.HomeNow();
												ELSE
													pressureBar.OpenJaw();
												END_IF
												IF IBD.homeRequired THEN
													IF NOT frontLoadPlate.enable THEN
														rearLoadPlate.moveToDischargePos();
													END_IF
													IBD.HomeNow();
												ELSE
													IBD.OpenIBD();
												END_IF
                                            	state.head := HEAD_STATES.Homing; 
											END_IF                             
    
    HEAD_STATES.Homing :                // 
											IF pressureBar.pressureBarOpen AND (NOT IBD.Ready OR NOT IBD.enable) THEN
                                                state.head := HEAD_STATES.HomingComplete;
																							
												IF motorizedSealFlatteners.sealFlattenersHorizontalAxisMotor.HomeRequired AND ((*motorizedSealFlatteners.enable*)HMIData.sealFlattenersInUse OR HMIData.sealAreaOptionSelection = (SealAreaOptionSelectionEnum.SealFlattenersWithPerfBreaker OR SealAreaOptionSelectionEnum.PerfBreaker)) AND pressureBar.jawClear   THEN
													motorizedSealFlatteners.sealFlattenersHorizontalAxisMotor.HomeNow();
													msfVerticalAxis.Retract();
													perfBreaker.MoveUp();
												END_IF	   
                                            END_IF
                                            
    HEAD_STATES.HomingComplete :            // 
											IF (NOT motorizedSealFlatteners.sealFlattenersHorizontalAxisMotor.HomeRequired) OR NOT motorizedSealFlatteners.enable THEN
												homeJawPB := FALSE;
												motorizedSealFlatteners.sealFlattenersVerticalAxis.Extend();
												state.head := HEAD_STATES.MovePassthrough;
											END_IF
                                           
    HEAD_STATES.MovePassthrough :           // 
                                            pressureBar.OpenJaw();
											IBD.OpenIBD();
                                            state.head := HEAD_STATES.MovingPassthrough;
    
    HEAD_STATES.MovingPassthrough :    		IF pressureBar.pressureBarOpen AND (IBD.IBDOpen OR HMIData.independentBagDeflatorSelection = BagDeflatorSelection.NotInstalled) THEN
                                                state.head := HEAD_STATES.MovedPassthrough;     
                                            END_IF
                                            
    HEAD_STATES.MovedPassthrough :          // 
                                            state.head := HEAD_STATES.Idle;
											setPassthroughPB := FALSE;
											//motorizedSealFlatteners.sealFlattenersHorizontalAxisMotor.MoveToPositionTorque(HMIData.bagWidth,1000,1000,1000,125);
											IF motorizedSealFlatteners.enable AND HMIData.sealFlattenersInUse THEN
												motorizedSealFlatteners.AutoMoveToStartPosition();
											ELSIF motorizedSealFlatteners.enable AND NOT HMIData.sealFlattenersInUse THEN
												motorizedSealFlatteners.AutoMoveToBagFeed();
                                            END_IF
                                                    
	HEAD_STATES.PrepareForAutomatedBagRemoval:
		//
		state.head := HEAD_STATES.PreparingForAutomatedBagRemoval;
		state.sb.automation := AUTOMATION_STATES.MoveSealFlattenersUp;
		
	HEAD_STATES.PreparingForAutomatedBagRemoval:
		//
		IF state.sb.automation = AUTOMATION_STATES.Done THEN
			_auxIOPhysical.ResetReadyForGrab();
			_auxIORemote.ResetReadyForGrab();
			state.head := HEAD_STATES.PreparedForAutomatedBagRemoval;
		END_IF
	
	HEAD_STATES.PreparedForAutomatedBagRemoval:
		//
		state.head := HEAD_STATES.Idle;
		state.sb.automation := AUTOMATION_STATES.Idle;
                                                    
    HEAD_STATES.Fault :                     hmiLight.TurnOff();
											HMIData.inCycle := FALSE;
											cycleTimer.IN := FALSE;
											bagDelivery.PointToPointOnFault();
											state.sb.sealSeparate := SEAL_SEPARATE_STATES.Idle;
											state.sb.releaseFeed := RELEASE_FEED_STATES.Idle;
											state.sb.openBag := BAG_OPEN_ASSIST_STATES.Idle;
											state.sb.finishCycle := FINISH_CYCLE_STATES.Idle;
											oVacOn := FALSE;
											filler.Reset();
											funnel.Reset();
											LPA.ManualOff();
											exitConveyorRun.Reset();
											externalExitConveyorRun.Reset();
											oRunPrinterRibbonUnwindMotor := FALSE;
											setPassthroughPB := FALSE;
											homeJawPB := FALSE;
											startCycle := FALSE;
											HMIData.initiateCycle := FALSE;
											factoryTestModeKeepCycling := FALSE;
											autoModeKeepCycling := FALSE;
											pressureBarCloseDelay.IN := FALSE;
											oSealBarExtend := FALSE;
											oSealBarRetract := TRUE;											
											posInhibit := FALSE;
											//perfBreaker.MoveUp();
											//msfVerticalAxis.Retract();
											
									
END_CASE

CASE state.sb.sealSeparate OF
	SEAL_SEPARATE_STATES.Shake:						
		//
		IF loadShelf.shakeStart = SHAKER_START_SELECTION.CycleStart OR
   		   loadShelf.shakeStart = SHAKER_START_SELECTION.Both THEN
		   loadShelf.Shake();
		END_IF
		
		//
		IF rearLoadPlate.shakeStart = SHAKER_START_SELECTION.CycleStart OR
   		   rearLoadPlate.shakeStart = SHAKER_START_SELECTION.Both THEN
		   rearLoadPlate.Shake();
		END_IF
		
		//
		IF frontLoadPlate.shakeStart = SHAKER_START_SELECTION.CycleStart OR
   		   frontLoadPlate.shakeStart = SHAKER_START_SELECTION.Both THEN
		   frontLoadPlate.Shake();
		END_IF

		//
		IF rearLoadPlate.Shaking OR frontLoadPlate.Shaking OR loadShelf.Shaking THEN
			state.sb.sealSeparate := SEAL_SEPARATE_STATES.Shaking;
		ELSIF enableIBDDeflate THEN
			state.sb.sealSeparate := SEAL_SEPARATE_STATES.BringInIBD;
		ELSE
			state.sb.sealSeparate := SEAL_SEPARATE_STATES.WaitForJawCloseDelay;
		END_IF
													
	SEAL_SEPARATE_STATES.Shaking:				    //
		IF NOT frontLoadPlate.Shaking AND NOT rearLoadPlate.Shaking AND NOT loadShelf.Shaking THEN
			state.sb.sealSeparate := SEAL_SEPARATE_STATES.PrepareToFeedToSeal;
		END_IF
		
	SEAL_SEPARATE_STATES.PrepareToFeedToSeal:
		IF HMIData.feedToSealInUse THEN
			IF enableBagOpen THEN
				bagOpenFingers.Release();
			END_IF
					motorizedSealFlatteners.AutoMovetoFeedToSeal();
					state.sb.sealSeparate := SEAL_SEPARATE_STATES.PreparingToFeedToSeal;	
		ELSE
			//
			IF enableIBDDeflate THEN
				state.sb.sealSeparate := SEAL_SEPARATE_STATES.BringInIBD;
			ELSE
				state.sb.sealSeparate := SEAL_SEPARATE_STATES.WaitForJawCloseDelay;
			END_IF	
		END_IF
	
	SEAL_SEPARATE_STATES.PreparingToFeedToSeal:
		IF motorizedSealFlatteners.state = SEAL_FLATTENER_STATES.Idle THEN
			state.sb.sealSeparate := SEAL_SEPARATE_STATES.PreparedToFeedToSeal;
		END_IF
	
	SEAL_SEPARATE_STATES.PreparedToFeedToSeal:
		state.sb.sealSeparate := SEAL_SEPARATE_STATES.FeedToSeal;

	SEAL_SEPARATE_STATES.FeedToSeal:
		IF HMIData.feedToSealInUse THEN
			bagDelivery.AutoFeedToSeal();
			state.sb.sealSeparate := SEAL_SEPARATE_STATES.FeedingToSeal;		
		ELSE
			//
			IF enableIBDDeflate THEN
				state.sb.sealSeparate := SEAL_SEPARATE_STATES.BringInIBD;
			ELSE
				state.sb.sealSeparate := SEAL_SEPARATE_STATES.WaitForJawCloseDelay;
			END_IF
		END_IF
	SEAL_SEPARATE_STATES.FeedingToSeal:
		//
		IF bagDelivery.state = BAG_DELIVERY_STATES.Ready THEN
			state.sb.sealSeparate := SEAL_SEPARATE_STATES.FedToSeal;
		END_IF
	
	SEAL_SEPARATE_STATES.FedToSeal:
		//
		// motorizedSealFlatteners.AutoEnableMotion();
		IF enableIBDDeflate THEN
			state.sb.sealSeparate := SEAL_SEPARATE_STATES.BringInIBD;
		ELSE
			state.sb.sealSeparate := SEAL_SEPARATE_STATES.WaitForJawCloseDelay;
		END_IF											
 
	SEAL_SEPARATE_STATES.BringInIBD: 				// Bring in IBD if enabled
													IF enableIBDDeflate THEN
														IBD.CloseIBD();
													END_IF 
													state.sb.sealSeparate := SEAL_SEPARATE_STATES.WaitForJawCloseDelay;
	
	SEAL_SEPARATE_STATES.WaitForJawCloseDelay: 	    // Wait for jaw close delay. 
													IF pressureBar.enable THEN
														LPA.ManualOff();
														pressureBarCloseDelay.IN := TRUE;
														IF (pressureBarCloseDelay.Q OR HMIData.pressureBarCloseDelay = 0) 
															//AND (funnel.closed OR NOT funnel.enable)
															THEN
															state.sb.sealSeparate := SEAL_SEPARATE_STATES.MoveJawIn;
															pressureBarCloseDelay.IN := FALSE;
														END_IF
                                                    ELSE 
                                                        state.sb.sealSeparate := SEAL_SEPARATE_STATES.ReverseBag;
                                                    END_IF
        
    SEAL_SEPARATE_STATES.MoveJawIn:                 // Perform actions as enabled - close jaw and move flatteners out. If jaw is disabled then go right to reverse bag
                                                    IF motorizedSealFlatteners.enable THEN
                                                        motorizedSealFlatteners.AutoMoveOut();
                                                    END_IF
                                                	sealTimer.IN := FALSE;
													pressureBar.CloseJaw();
                                                    state.sb.sealSeparate := SEAL_SEPARATE_STATES.MovingJawIn;
                                                    
    SEAL_SEPARATE_STATES.MovingJawIn :              // If Jaw is in and flatteners out then move on
                                                    IF (motorizedSealFlatteners.state = SEAL_FLATTENER_STATES.MovedFlattenersOut OR NOT motorizedSealFlatteners.enable)
														OR  (motorizedSealFlatteners.state = SEAL_FLATTENER_STATES.Idle AND MSFatBagFeedSetpoint)
                                                        AND (pressureBar.clamped OR NOT pressureBar.enable)
                                                        THEN
                                                            state.sb.sealSeparate := SEAL_SEPARATE_STATES.MovedJawIn;    
                                                    END_IF
                                                                
    SEAL_SEPARATE_STATES.MovedJawIn :               // Will add sealing logic here
													IF iJawClampsRetracted OR NOT pressureBar.enable THEN
                                                    	state.sb.sealSeparate := SEAL_SEPARATE_STATES.ReverseBag;
                                                    END_IF
													
    SEAL_SEPARATE_STATES.ReverseBag :               // Reverse bag if bag delivery enabled, otherwise open jaw
													//IBD.OpenFull();
                                                    IF bagDelivery.enable THEN
                                                        bagDelivery.AutoReverseBag();
                                                        state.sb.sealSeparate := SEAL_SEPARATE_STATES.ReversingBag;
                                                    ELSE state.sb.sealSeparate := SEAL_SEPARATE_STATES.Done;    
                                                    END_IF
                                                                    
    SEAL_SEPARATE_STATES.ReversingBag :             // 
													
													IF NOT HMIData.separateBeforeSeal THEN
														sealTimer.PT := TO_TIME(HMIData.sealBarDwell * 1000);
														sealTimer.IN := TRUE;
														IF NOT sealTimer.Q THEN
															oSealBarExtend := TRUE; 
															oSealBarRetract := FALSE;															
														ELSE 
															oSealBarExtend := FALSE;
															oSealBarRetract := TRUE;
														END_IF
													END_IF

                                                    IF ((motorizedSealFlatteners.state = SEAL_FLATTENER_STATES.MovedFlattenersOut OR NOT motorizedSealFlatteners.enable)
														OR  (motorizedSealFlatteners.state = SEAL_FLATTENER_STATES.Idle AND MSFatBagHoldSetpoint)//MSFatBagFeedSetpoint)
                                                        AND (pressureBar.clamped OR NOT pressureBar.enable)
                                                        AND (bagDelivery.state = BAG_DELIVERY_STATES.ReverseDone OR NOT bagDelivery.enable))
														AND (sealTimer.Q OR HMIData.separateBeforeSeal)
                                                        THEN
															IF NOT HMIData.separateBeforeSeal THEN
																HMIData.sealBarCycles.Increment();
															END_IF
															
															sealTimer.IN := FALSE;
                                                            state.sb.sealSeparate := SEAL_SEPARATE_STATES.Reversedbag;
                                                    END_IF
													
    SEAL_SEPARATE_STATES.Reversedbag :              // 
													//Print mid cycle if needed.
													IF zebraPrinter.enable AND HMIData.printerCycleSelection = PrinterCycleSelection.PrintMidCycle THEN
														state.sb.printOutOfCycle := PRINT_OUT_OF_CYCLE_STATES.WaitForPrinter;
													END_IF
													
                                                    state.sb.sealSeparate := SEAL_SEPARATE_STATES.SealBag;
													
	SEAL_SEPARATE_STATES.SealBag:					
													sealTimer.IN := TRUE;
													IF HMIData.separateBeforeSeal THEN														
														sealTimer.PT := TO_TIME(HMIData.sealBarDwell * 1000);
														sealTimer.IN := TRUE;
														IF NOT sealTimer.Q THEN
															oSealBarExtend := TRUE;
															oSealBarRetract := FALSE;
														ELSE 
															sealTimer.IN := FALSE;
															oSealBarExtend := FALSE;
															oSealBarRetract := TRUE;
															HMIData.sealBarCycles.Increment();
															state.sb.sealSeparate := SEAL_SEPARATE_STATES.Done;
														END_IF
													ELSE			
														state.sb.sealSeparate := SEAL_SEPARATE_STATES.Done;
													END_IF                      
    SEAL_SEPARATE_STATES.Done:    
													                    //
    SEAL_SEPARATE_STATES.Fault:						//
END_CASE

_waitForPressureBarOpenDelay(IN := state.sb.releaseFeed = RELEASE_FEED_STATES.WaitForPressureBarOpenTimer, PT := TO_TIME((HMIData.pressureBarOpenDelay * 1000.0)));

CASE state.sb.releaseFeed OF
    RELEASE_FEED_STATES.Idle :  
                      //
    
	RELEASE_FEED_STATES.WaitForPressureBarOpenTimer : 		// Adding in Jaw Open Delay
													IF _waitForPressureBarOpenDelay.Q THEN
														state.sb.releaseFeed := RELEASE_FEED_STATES.MoveJawOutAndDropBag;
													END_IF
													

                                                   
    RELEASE_FEED_STATES.MoveJawOutAndDropBag :        // 
                                                    IF (motorizedSealFlatteners.state = SEAL_FLATTENER_STATES.MovedFlattenersOut OR NOT motorizedSealFlatteners.enable)
														OR (motorizedSealFlatteners.state = SEAL_FLATTENER_STATES.Idle AND MSFatBagFeedSetpoint)
                                                        AND (pressureBar.clamped OR NOT pressureBar.enable)
                                                        AND ((bagDelivery.state = BAG_DELIVERY_STATES.ReverseDone) OR HMIData.enableDryCycle)
                                                        OR (bagDelivery.state =  BAG_DELIVERY_STATES.WaitingForPrinter AND zebraPrinter.enable)
                                                        OR NOT bagDelivery.enable
                                                        THEN
                                                            IF (*motorizedSealFlatteners.enable*)HMIData.sealFlattenersInUse THEN
                                                                motorizedSealFlatteners.AutoMoveToClearance();
																//motorizedSealFlatteners.AutoMoveToBagHolding();
                                                            ELSIF (HMIData.mailerMaterial = MAILER_MATERIAL.paper) THEN
																perfBreaker.Retract(); 
                                                            END_IF
                                                            
                                                            IF enableBagOpen THEN
                                                                pressureBar.OpenJawForBagFeed();
															ELSE
																pressureBar.OpenJaw();
                                                            END_IF
															
                                                            //IBD.OpenFull();
// 															IF enableBagOpen THEN
// 																bagOpenFingers.Release();
// 															END_IF
															
															IF enableIBDEject THEN
																IBD.CloseIBD();
															END_IF
															
															IF rearLoadPlate.enable THEN
																rearLoadPlate.Trigger();
															END_IF
															
															IF frontLoadPlate.enable THEN
																frontLoadPlate.Trigger();
															END_IF
															
															IF loadShelf.enable THEN
																loadShelf.Trigger();
															END_IF
														
															IF TO_DINT(HMIData.exitConveyorDwell) <> 0 THEN
																exitConveyorRun.Trigger();
															END_IF
															
															IF TO_DINT(HMIData.externalExitConveyorDwell) <> 0 AND NOT printAndApply.enable THEN
																externalExitConveyorRun.Trigger();
															END_IF
															
															IF HMIData.lpaBagEjectAssistEnable THEN
																LPA.ManualOn();
															END_IF
															IBD.OpenFull();
                                                           bagDropTimer.IN := TRUE;
														   state.sb.releaseFeed := RELEASE_FEED_STATES.MovingJawOutAndDroppingBag;
                                                    END_IF
													
	 RELEASE_FEED_STATES.MovingJawOutAndDroppingBag :
														// If printer is enabled then perform printer operation of bag delivery, otherwise just feed new bag out.
                                                        // In the case that bagDelivery is disabled then we're done with release and feed
														IF (motorizedSealFlatteners.state = SEAL_FLATTENER_STATES.MovedFlattenersOut 
														OR MSFatOutSetpoint OR MSFatBagFeedSetpoint) 
														AND (*motorizedSealFlatteners.enable*)HMIData.sealFlattenersInUse THEN
															motorizedSealFlatteners.AutoMoveToClearance();														 
														END_IF

														IF enableBagOpen AND pressureBar.actualPosition >= 0.5 THEN
 															bagOpenFingers.Release();
 														END_IF	
														
                                                        IF bagDropTimer.Q 
															AND (perfBreaker.retractedStatus OR NOT (HMIData.mailerMaterial = MAILER_MATERIAL.paper))
															AND (motorizedSealFlatteners.state = SEAL_FLATTENER_STATES.MovedFlattenersToBagFeed OR MSFatBagFeedSetpoint OR NOT motorizedSealFlatteners.enable )
															THEN   

															
															
															IF bagDelivery.enable AND NOT (zebraPrinter.enable) THEN // No Print Required
																bagDropTimer.IN := FALSE;
																bagDelivery.AutoFeedBagOut();
 																LPA.ManualOff();
                                                                state.sb.releaseFeed := RELEASE_FEED_STATES.MovingJawOutAndFeedingBag;
                                                            ELSIF (bagDelivery.enable AND zebraPrinter.enable) THEN // Print Required
																IF HMIData.printerCycleSelection = PrinterCycleSelection.PrintWhileFeeding THEN
																	bagDropTimer.IN := FALSE;
																	bagDelivery.AutoWaitForPrinter();
																	LPA.ManualOff();
																	state.sb.releaseFeed := RELEASE_FEED_STATES.WaitForPrinter;
																ELSIF HMIData.printerCycleSelection = PrinterCycleSelection.PrintMidCycle THEN
																	
																	 IF state.sb.printOutOfCycle = PRINT_OUT_OF_CYCLE_STATES.Done THEN
																		bagDropTimer.IN := FALSE;
																		bagDelivery.AutoFeedBagOut();
																		LPA.ManualOff();
																		state.sb.releaseFeed := RELEASE_FEED_STATES.MovingJawOutAndFeedingBag;
																	 END_IF
																ELSE
																	bagDropTimer.IN := FALSE;
																	bagDelivery.AutoFeedBagOut();
																	LPA.ManualOff();
																	state.sb.releaseFeed := RELEASE_FEED_STATES.MovingJawOutAndFeedingBag;
																END_IF
                                                                

                                                            ELSE 
                                                                state.sb.releaseFeed := RELEASE_FEED_STATES.Done;
                                                            END_IF												
    													END_IF
														
    RELEASE_FEED_STATES.WaitForPrinter :            // Data Ready means the printer has a label and we're all set to print
                                                    IF zebraPrinter.state = PRINTER_STATES.DataReady THEN
                                                        IF HMIData.lpaDuringBagFeedEnable THEN
                                                            LPA.ManualOn();
                                                        END_IF														
                                                        state.sb.releaseFeed := RELEASE_FEED_STATES.FeedToOffset;
                                                    END_IF
													IF enableBagOpen AND pressureBar.actualPosition >= 0.5 THEN
 														bagOpenFingers.Release();
 													END_IF	
                                                    
    RELEASE_FEED_STATES.FeedToOffset :              // This starts feeding to the print offset
													IF (motorizedSealFlatteners.state = SEAL_FLATTENER_STATES.MovedFlattenersToBagFeed OR NOT motorizedSealFlatteners.enable OR MSFatBagFeedSetpoint) THEN
														bagDelivery.AutoPrinterReady();
                                                    	state.sb.releaseFeed := RELEASE_FEED_STATES.FeedingToOffset;
													END_IF
													IF enableBagOpen AND pressureBar.actualPosition >= 0.5 THEN
 														bagOpenFingers.Release();
 													END_IF	
                                                    
                                                        
    RELEASE_FEED_STATES.FeedingToOffset :            // Once offset done start printing
													IF HMIData.printOutOfCycleEnable THEN
														IF bagDelivery.state = BAG_DELIVERY_STATES.CreatedSlack THEN  
															state.sb.releaseFeed := RELEASE_FEED_STATES.StartPrinting;
														END_IF     
													ELSE
														IF bagDelivery.state = BAG_DELIVERY_STATES.FedToPrintOffset THEN  
															state.sb.releaseFeed := RELEASE_FEED_STATES.StartPrinting;
														END_IF     
													END_IF  
														IF enableBagOpen AND pressureBar.actualPosition >= 0.5 THEN
															bagOpenFingers.Release();
														END_IF	                                     
    
    RELEASE_FEED_STATES.StartPrinting :             // Printer starts print cycle and bag delivery starts moving at print speed
													zebraPrinter.AutoPrintNow();
                                                    state.sb.releaseFeed := RELEASE_FEED_STATES.SendPrintSignal;                                            

    RELEASE_FEED_STATES.SendPrintSignal:            // 
              
													IF enableBagOpen AND pressureBar.actualPosition >= 0.5 THEN
 														bagOpenFingers.Release();
 													END_IF	
													IF zebraPrinter.printHeadDebounced THEN
														bagDelivery.AutoStartPrintFeed();
														zebraPrinter.AutoSendPrintSignal();
														barcodeVerifier.Trigger();
                                                        state.sb.releaseFeed := RELEASE_FEED_STATES.Printing;
                                                    END_IF                                        

    RELEASE_FEED_STATES.Printing :                // 
													IF enableBagOpen AND pressureBar.actualPosition >= 0.5 THEN
 														bagOpenFingers.Release();
 													END_IF	
                                                    IF zebraPrinter.state = PRINTER_STATES.DonePrinting THEN
                                                        state.sb.releaseFeed := RELEASE_FEED_STATES.StopPrinting;
                                                    END_IF
                                                    
    RELEASE_FEED_STATES.StopPrinting :                // Tell bag delivery it's okay to feed out the rest of the bag and the printer that it can prep itself for the next print
                                                    bagDelivery.AutoPrinterDone();
                                                    zebraPrinter.AutoAckPrintDone();
                                                    state.sb.releaseFeed := RELEASE_FEED_STATES.MovingJawOutAndFeedingBag;
                                                                                                            
    RELEASE_FEED_STATES.MovingJawOutAndFeedingBag :    // 
													
													IF enableBagOpen AND pressureBar.actualPosition >= 0.5 THEN
 														bagOpenFingers.Release();
 													END_IF
													IF (bagDelivery.state = BAG_DELIVERY_STATES.Ready OR NOT bagDelivery.enable)
                                                        AND (motorizedSealFlatteners.state = SEAL_FLATTENER_STATES.MovedFlattenersToBagFeed OR NOT motorizedSealFlatteners.enable OR NOT HMIData.sealFlattenersInUse) 
                                                        AND (pressureBar.pressureBarOpen OR NOT pressureBar.enable)
														
                                                        THEN
                                                            state.sb.releaseFeed := RELEASE_FEED_STATES.MovedJawOutAndFedBag;
                                                    END_IF
                                                    
    RELEASE_FEED_STATES.MovedJawOutAndFedBag :      // Wait until bag is fed out before triggering barcode fail.
													IF barcodeVerifier.barcodeFault THEN
														barcodeVerificationFailed.Trigger();
													END_IF 
													
													// Trigger end cycle print
													IF HMIData.printerCycleSelection = PrinterCycleSelection.PrintEndCycle THEN
														state.sb.printOutOfCycle := PRINT_OUT_OF_CYCLE_STATES.WaitForPrinter;
													END_IF
													
													IF enableIBDDeflate OR enableIBDEject THEN
														IBD.OpenIBD();
													END_IF
													state.sb.releaseFeed := RELEASE_FEED_STATES.Done;
													
													IF HPA.DwellSetting <> 0 THEN
														HPA.Trigger();	
													END_IF	 
													
    RELEASE_FEED_STATES.Done :						//
    RELEASE_FEED_STATES.Fault :						//
END_CASE

CASE state.sb.openBag OF
    BAG_OPEN_ASSIST_STATES.Idle:                    // 
                                                    bagOpenCheckDelay.IN := FALSE;
                                                                         
    BAG_OPEN_ASSIST_STATES.MoveJawIn :              // Close jaw against bag. In the future we may also start vacuum here
                                                    pressureBar.CloseJawNoLatch();
												
													
													//oVacOn := TRUE; // Hard coded for now, this is vacuum
                                                    state.sb.openBag := BAG_OPEN_ASSIST_STATES.MovingJawIn;        
                                                    
    BAG_OPEN_ASSIST_STATES.MovingJawIn :            // Move on once jaw is closed
                                                    IF pressureBar.iPressureBarClosed OR NOT pressureBar.enable THEN
                                                        state.sb.openBag := BAG_OPEN_ASSIST_STATES.MovedJawIn;        
                                                    END_IF
                                                    
    BAG_OPEN_ASSIST_STATES.MovedJawIn :             // Hold onto the bag with vacuum to build suction
													IF HMIData.mailerMaterial = MAILER_MATERIAL.paper THEN
														perfBreaker.MoveDown();
													END_IF	
													
													IF HMIData.enableDryCycle THEN
														state.sb.openBag := BAG_OPEN_ASSIST_STATES.MoveJawOut;
													ELSE
														vacuumHoldTimer.IN := TRUE;
														oVacOn := TRUE; // Hard coded for now, this is vacuum
														IF vacuumHoldTimer.Q THEN
															vacuumHoldTimer.IN := FALSE;
															state.sb.openBag := BAG_OPEN_ASSIST_STATES.MoveJawOut;
														END_IF            
													END_IF
                                                                   
    BAG_OPEN_ASSIST_STATES.MoveJawOut :             // Open the jaw and move seal flatteners in and to bag holding
                                                    (*IF HMIData.enablePerfBreaker AND NOT (*motorizedSealFlatteners.enable*)HMIData.sealFlattenersInUse  THEN
														perfBreaker.Extend();
													END_IF*)
													pressureBar.OpenJaw();
													IF HMIData.mailerMaterial = MAILER_MATERIAL.poly THEN
														motorizedSealFlatteners.AutoMoveIn();
													END_IF
                                                    state.sb.openBag := BAG_OPEN_ASSIST_STATES.MovingJawOutAndGrab;
                                                                                             
    BAG_OPEN_ASSIST_STATES.MovingJawOutAndGrab :    // Once everything that is enabled is homed finish cycle 
													IF pressureBar.actualPosition > grabDistance THEN
													bagOpenFingers.Grab();
													bagOpenFingerDelay.IN := FALSE;
													state.sb.openBag := BAG_OPEN_ASSIST_STATES.CheckForSuccessfulBagGrab;	
													END_IF
													
													(*bagOpenFingerDelay.IN := TRUE;
													IF bagOpenFingerDelay.Q THEN
														bagOpenFingers.Grab();
														bagOpenFingerDelay.IN := FALSE;
														state.sb.openBag := BAG_OPEN_ASSIST_STATES.CheckForSuccessfulBagGrab;
													END_IF*)
													  

	BAG_OPEN_ASSIST_STATES.CheckForSuccessfulBagGrab : 	//
														IF bagOpenRetryCount < bagOpenRetrySetting THEN
															bagOpenCheckDelay.IN := TRUE;
															IF bagOpenCheckDelay.Q THEN
																IF bagOpenFingers.CheckIfBagGrabbed(TRUE) OR HMIData.enableDryCycle THEN // This method checks to see if the bag is grabbed and returns true if so.
																	IF HMIData.mailerMaterial = MAILER_MATERIAL.paper THEN
																		 motorizedSealFlatteners.AutoMoveIn();
																	END_IF
																	state.sb.openBag := BAG_OPEN_ASSIST_STATES.OpenBag;
																ELSE 
																	state.sb.openBag := BAG_OPEN_ASSIST_STATES.BagFailedToOpen;
																END_IF
																bagOpenCheckDelay.IN := FALSE;
															END_IF
														ELSE 
															motorizedSealFlatteners.AutoMoveToBagHolding();
															state.sb.openBag := BAG_OPEN_ASSIST_STATES.MovingJawOutAfterGrab;
														END_IF
													  
	BAG_OPEN_ASSIST_STATES.BagFailedToOpen :			//
													IF (HMIData.mailerMaterial = MAILER_MATERIAL.paper) AND HMIData.enablePaperBagger THEN
														//perfBreaker.MoveDown();
													END_IF 
														bagOpenFingers.Release();
														bagOpenRetryCount := bagOpenRetryCount + 1;
														IF bagOpenRetryCount < bagOpenRetrySetting THEN
															state.sb.openBag := BAG_OPEN_ASSIST_STATES.MoveJawIn;
														ELSIF HMIData.bagOpenFeedNewBagCount < HMIData.bagOpenFeedNewBagSetting THEN
															HMIData.bagOpenFeedNewBagCount := HMIData.bagOpenFeedNewBagCount + 1;
															bagOpenRetryCount := 0;
															motorizedSealFlatteners.AutoMoveOut();
															oVacOn := FALSE;
															state.sb.openBag := BAG_OPEN_ASSIST_STATES.FeedNewBag;
															
														ELSE 
															//IF (motorizedSealFlatteners.state = SEAL_FLATTENER_STATES.Idle OR NOT motorizedSealFlatteners.enable) THEN
																motorizedSealFlatteners.AutoMoveToBagHolding();
																bagFailedToOpen.Trigger();
																
																state.sb.openBag := BAG_OPEN_ASSIST_STATES.MovingJawOutAfterGrab;
																bagOpenRetryCount := 0; 
																HMIData.bagOpenFeedNewBagCount := 0;
																HMIData.bagsRejectedTotal.Increment();
																Globals.rejectedBagCount := Globals.rejectedBagCount + 1;
															//END_IF
															
														END_IF
	
	BAG_OPEN_ASSIST_STATES.OpenBag :					//													
														// Move flatteners now if no funnel. Otherwise let the funnel move the flatteners when done
														IF MSFatInSetpoint AND NOT funnel.enable THEN 
															motorizedSealFlatteners.AutoMoveToBagHolding();
														END_IF
														
                                                    	IF //MSFatBagHoldSetpoint THEN
														(motorizedSealFlatteners.state = SEAL_FLATTENER_STATES.MovingFlattenersDown) OR NOT HMIData.sealFlattenersInUse THEN
															state.sb.openBag := BAG_OPEN_ASSIST_STATES.bagOpening; 
														END_IF
														
	BAG_OPEN_ASSIST_STATES.BagOpening :					//
																												
                                                    	//IF MSFatBagHoldSetpoint THEN
															state.sb.openBag := BAG_OPEN_ASSIST_STATES.bagOpened; 
														//END_IF
														
														
	BAG_OPEN_ASSIST_STATES.BagOpened :
															bagOpened := TRUE;
														// Move flatteners now if no funnel. Otherwise let the funnel move the flatteners when done
																										
                                                    	//IF MSFatBagHoldSetpoint THEN
															bagOpenRetryCount := 0;
															HMIData.bagOpenFeedNewBagCount := 0;														
															state.sb.openBag := BAG_OPEN_ASSIST_STATES.MovingJawOutAfterGrab; 
														//END_IF
														
    BAG_OPEN_ASSIST_STATES.MovingJawOutAfterGrab :		// 
														IF (pressureBar.pressureBarOpen OR NOT pressureBar.enable) 
															AND ((motorizedSealFlatteners.state = SEAL_FLATTENER_STATES.Idle OR NOT motorizedSealFlatteners.enable)
																OR (motorizedSealFlatteners.state = SEAL_FLATTENER_STATES.MovedFlattenersIn AND HMIData.funnelFactorySelection = FunnelSelection.BagLoadingTray))
															THEN
																state.sb.openBag := BAG_OPEN_ASSIST_STATES.MovedJawOut;        
														END_IF	 
														
	BAG_OPEN_ASSIST_STATES.MovedJawOut :                // 
														oVacOn := FALSE; 		// Hard coded for now, this is vacuum
														state.sb.openBag := BAG_OPEN_ASSIST_STATES.Done;
                               
	BAG_OPEN_ASSIST_STATES.FeedNewBag :   			//
													IF (motorizedSealFlatteners.state = SEAL_FLATTENER_STATES.Idle OR NOT motorizedSealFlatteners.enable) THEN
														state.head := HEAD_STATES.SealAndSeparateBag;
													END_IF
										                        
    BAG_OPEN_ASSIST_STATES.Done:                    //                                             
    BAG_OPEN_ASSIST_STATES.Fault:                   //
													

END_CASE

CASE state.sb.finishCycle OF
	FINISH_CYCLE_STATES.Start :								//
															IF funnel.enable THEN
																state.sb.finishCycle := FINISH_CYCLE_STATES.OpenFunnel;
															ELSIF enableBagOpen THEN
																state.sb.finishCycle := FINISH_CYCLE_STATES.Shake;
															ELSE
																IF motorizedSealFlatteners.enable THEN
																	state.sb.finishCycle := FINISH_CYCLE_STATES.BringSealFlattenersInAndDown;
																ELSE
																	state.sb.finishCycle := FINISH_CYCLE_STATES.Shake;
																END_IF
															END_IF
															LPA.DwellSetting := TO_DINT(HMIData.lpaDwell * 1000);
															IF LPA.DwellSetting <> 0 THEN
																LPA.Trigger();
															END_IF
	
	FINISH_CYCLE_STATES.OpenFunnel :						//
															LPA.DwellSetting := TO_DINT(HMIData.lpaDwell * 1000);
															IF LPA.DwellSetting <> 0 THEN
																LPA.Trigger();
															END_IF
															motorizedSealFlatteners.AutoMoveToBagHolding();
															funnel.Open();
															state.sb.finishCycle := FINISH_CYCLE_STATES.OpeningFunnel;
	
	FINISH_CYCLE_STATES.OpeningFunnel :						//
															IF funnel.opened THEN
																state.sb.finishCycle := FINISH_CYCLE_STATES.OpenedFunnel;
															END_IF
	
	FINISH_CYCLE_STATES.OpenedFunnel :						//
															//IF enableBagOpen THEN
															IF iLeftFingerBagPresent AND iRightFingerBagPresent THEN
																	//IF motorizedSealFlatteners.enable THEN
																	//	state.sb.finishCycle := FINISH_CYCLE_STATES.BringSealFlattenersToBagHolding;
																	//ELSE
																		
																		state.sb.finishCycle := FINISH_CYCLE_STATES.Shake;
																	//END_IF
																	bagOpened := TRUE;
																ELSE
																	IF bagOpenRetryCount < bagOpenRetrySetting THEN
																		funnel.Close();
																		bagOpenRetryCount := bagOpenRetryCount + 1;
																		state.sb.finishCycle := FINISH_CYCLE_STATES.ClosingFunnelForRetry;
																	ELSE
																		funnel.Close();
																		bagOpenRetryCount := 0;
																		bagFailedToOpen.Trigger();
																		HMIData.bagsRejectedTotal.Increment();
																		state.sb.finishCycle := FINISH_CYCLE_STATES.Shake;
																	END_IF
																END_IF
															
																
															//END_IF
	
	FINISH_CYCLE_STATES.ClosingFunnelForRetry :				//
															IF funnel.closed THEN
																state.sb.finishCycle := FINISH_CYCLE_STATES.Start;
															END_IF												
	
	FINISH_CYCLE_STATES.BringSealFlattenersInAndDown :		//
															motorizedSealFlatteners.AutoMoveToHandLoad();
															state.sb.finishCycle := FINISH_CYCLE_STATES.BringingSealFlattenersInAndDown;
	
	FINISH_CYCLE_STATES.BringingSealFlattenersInAndDown :	//
															IF motorizedSealFlatteners.state = SEAL_FLATTENER_STATES.Idle THEN
																state.sb.finishCycle := FINISH_CYCLE_STATES.SealFlattenersInAndDown;
															END_IF
	
	FINISH_CYCLE_STATES.SealFlattenersInAndDown :			//
															state.sb.finishCycle := FINISH_CYCLE_STATES.Shake;
	
	FINISH_CYCLE_STATES.BringSealFlattenersToBagHolding:	//
															motorizedSealFlatteners.AutoMoveToBagHolding();
															state.sb.finishCycle := FINISH_CYCLE_STATES.BringingSealFlattenersToBagHolding;
	
	FINISH_CYCLE_STATES.BringingSealFlattenersToBagHolding: //
															IF motorizedSealFlatteners.state = SEAL_FLATTENER_STATES.Idle THEN
																state.sb.finishCycle := FINISH_CYCLE_STATES.SealFlattenersAtBagHolding;
															END_IF
																
	FINISH_CYCLE_STATES.SealFlattenersAtBagHolding : 		//
															state.sb.finishCycle := FINISH_CYCLE_STATES.Shake;
															
	FINISH_CYCLE_STATES.Shake:
		//
		IF loadShelf.shakeStart = SHAKER_START_SELECTION.BagOpen OR
   		   loadShelf.shakeStart = SHAKER_START_SELECTION.Both THEN
		   loadShelf.Shake();
		END_IF
		
		//
		IF rearLoadPlate.shakeStart = SHAKER_START_SELECTION.BagOpen OR
   		   rearLoadPlate.shakeStart = SHAKER_START_SELECTION.Both THEN
		   rearLoadPlate.Shake();
		END_IF
		
		//
		IF frontLoadPlate.shakeStart = SHAKER_START_SELECTION.BagOpen OR
   		   frontLoadPlate.shakeStart = SHAKER_START_SELECTION.Both THEN
		   frontLoadPlate.Shake();
		END_IF

		IF rearLoadPlate.Shaking OR frontLoadPlate.Shaking OR loadShelf.Shaking THEN
			state.sb.finishCycle := FINISH_CYCLE_STATES.Shaking;
		ELSIF zebraPrinter.enable AND HMIData.printerCycleSelection <> PrinterCycleSelection.PrintWhileFeeding THEN
			state.sb.finishCycle := FINISH_CYCLE_STATES.WaitForOutOfCyclePrint;
		ELSE
			state.sb.finishCycle := FINISH_CYCLE_STATES.Done;
		END_IF
	
	FINISH_CYCLE_STATES.Shaking:
		IF NOT frontLoadPlate.Shaking AND NOT rearLoadPlate.Shaking AND NOT loadShelf.Shaking THEN
			IF zebraPrinter.enable AND HMIData.printerCycleSelection <> PrinterCycleSelection.PrintWhileFeeding THEN
				state.sb.finishCycle := FINISH_CYCLE_STATES.WaitForOutOfCyclePrint;
			ELSE
				state.sb.finishCycle := FINISH_CYCLE_STATES.Done;
			END_IF
		END_IF	
	
	FINISH_CYCLE_STATES.WaitForOutOfCyclePrint:
		//
		IF bagOpened THEN
        	IF NOT bagOpenFingers.CheckIfBagGrabbed(FALSE) AND NOT HMIData.enableDryCycle THEN
				openedBagWasRemoved.Trigger();
				bagOpened := FALSE;
			END_IF
		END_IF
		
		IF state.sb.printOutOfCycle = PRINT_OUT_OF_CYCLE_STATES.Done THEN
			state.sb.printOutOfCycle := PRINT_OUT_OF_CYCLE_STATES.Idle;
			state.sb.finishCycle := FINISH_CYCLE_STATES.Done;
		END_IF	
	
	FINISH_CYCLE_STATES.Done :								
		//
		bagOpenRetryCount := 0;
END_CASE

_waitForSealFlattenersUpTimer(IN := state.sb.automation = AUTOMATION_STATES.MovingSealFlattenersUp);
CASE state.sb.automation OF
	
	AUTOMATION_STATES.MoveSealFlattenersUp:
		motorizedSealFlatteners.sealFlattenersVerticalAxis.Retract();
		state.sb.automation := AUTOMATION_STATES.MovingSealFlattenersUp;
		
	AUTOMATION_STATES.MovingSealFlattenersUp:	
		IF _waitForSealFlattenersUpTimer.Q THEN
			motorizedSealFlatteners.AutoMoveOut();
			state.sb.automation := AUTOMATION_STATES.MovingSealFlattenersOut;
		END_IF
		
	AUTOMATION_STATES.MoveSealFlattenersOut:	
		motorizedSealFlatteners.AutoMoveOut();
		state.sb.automation := AUTOMATION_STATES.MoveSealFlattenersOut;
	
	AUTOMATION_STATES.MovingSealFlattenersOut:
		IF motorizedSealFlatteners.state = SEAL_FLATTENER_STATES.MovedFlattenersOut THEN
			motorizedSealFlatteners.Reset();
			state.sb.automation := AUTOMATION_STATES.MovedSealFlattenersIn;
		END_IF
		
	AUTOMATION_STATES.MovedSealFlattenersIn:
		state.sb.automation := AUTOMATION_STATES.DisableBagOpenSensing;
	
	AUTOMATION_STATES.DisableBagOpenSensing:
		bagOpened := FALSE;
		state.sb.automation := AUTOMATION_STATES.RaiseBOF;	
	
	AUTOMATION_STATES.RaiseBOF:
		bagOpenFingers.Release();
		state.sb.automation := AUTOMATION_STATES.Done; 
END_CASE

// Print out of cycle
_waitForTakeupTimer(IN := state.sb.printOutOfCycle = PRINT_OUT_OF_CYCLE_STATES.WaitForTakeup);
CASE state.sb.printOutOfCycle OF
	PRINT_OUT_OF_CYCLE_STATES.Idle:
		// Machine state machine will start this sub state by setting to "WaitForPrinter"
		
	PRINT_OUT_OF_CYCLE_STATES.WaitForPrinter:
		// Wait for label
		IF zebraPrinter.state = PRINTER_STATES.DataReady THEN
        	state.sb.printOutOfCycle := PRINT_OUT_OF_CYCLE_STATES.StartPrinting;
        END_IF
		
	PRINT_OUT_OF_CYCLE_STATES.StartPrinting:
		// Turn off power to rear motor and disable tension fault. Tell Zebra FB to prep for print cycle.
		zebraPrinter.AutoPrintNow();
		bagDelivery.bagFeedRearMotor.SetTorque(0);
		bagDelivery.bagFeedRearMotor.DisableTensionFault();
        state.sb.printOutOfCycle := PRINT_OUT_OF_CYCLE_STATES.SendPrintSignal;
	
	PRINT_OUT_OF_CYCLE_STATES.SendPrintSignal:
		// After print head and compensator are down, send the print and start barcode verifier
		IF zebraPrinter.printHeadDebounced THEN												
			zebraPrinter.AutoSendPrintSignal();
			barcodeVerifier.Trigger();
			state.sb.printOutOfCycle := PRINT_OUT_OF_CYCLE_STATES.Printing;
        END_IF
													
	PRINT_OUT_OF_CYCLE_STATES.Printing:
		// Wait for print to complete
		 IF zebraPrinter.state = PRINTER_STATES.DonePrinting THEN
         	state.sb.printOutOfCycle := PRINT_OUT_OF_CYCLE_STATES.FinishedPrinting;
         END_IF
		 
	PRINT_OUT_OF_CYCLE_STATES.FinishedPrinting:
		// All done. Tell Zebra FB that we see it finished, and up the torque on the rear motor to take up slack
		zebraPrinter.AutoAckPrintDone();
		bagDelivery.bagFeedRearMotor.SetTorque(100);
        state.sb.printOutOfCycle := PRINT_OUT_OF_CYCLE_STATES.WaitForTakeup;
		
	PRINT_OUT_OF_CYCLE_STATES.WaitForTakeup:
		// Change this to a rear motor move in reverse to take up faster?
		IF  _waitForTakeupTimer.Q THEN
			bagDelivery.bagFeedRearMotor.EnableTensionFault();
			//bagDelivery._bagFeedRearMotor.SetTorque((TO_DINT(HMIData.bagTensionSetting * 100)));
		END_IF
		state.sb.printOutOfCycle := PRINT_OUT_OF_CYCLE_STATES.Done;
		
	PRINT_OUT_OF_CYCLE_STATES.Done:
		// Machine state machine will set this back to idle.
		
	PRINT_OUT_OF_CYCLE_STATES.Fault:
		//
		
END_CASE

HMIData.initiateCycle := FALSE;

END_FUNCTION_BLOCK

// FBs/Recipie Manangment/RecallValues
FUNCTION RecallValues : DWORD
VAR
	recipieManager : Recipe_Management.RecipeManCommands;
	recipeName : STRING;
	recResult : UDINT;
END_VAR

recResult := recipieManager.CreateRecipe(RecipeDefinitionName := 'Recipes', RecipeName := 'Automatic');
recResult := recipieManager.GetRecipeNames('Recipes', ADR(recipeName),1,0);
recResult := recipieManager.LoadAndWriteRecipe(RecipeDefinitionName := 'Recipes', RecipeName := 'Automatic');

IF HMIData.bagsMade.count = 0 THEN
	recResult := recipieManager.CreateRecipe(RecipeDefinitionName := 'Recipes', RecipeName := 'Periodic');
	recResult := recipieManager.GetRecipeNames('Recipes', ADR(recipeName),1,0);
	recResult := recipieManager.LoadAndWriteRecipe(RecipeDefinitionName := 'Recipes', RecipeName := 'Periodic');
END_IF

END_FUNCTION

// FBs/Recipie Manangment/SaveValues
FUNCTION SaveValues : DWORD
VAR
	recipieManager : Recipe_Management.RecipeManCommands;
	recipeName : STRING;
	recResult : DWORD;
END_VAR

IF HMIData.bagsMade.count <> 0 THEN
	recResult := recipieManager.CreateRecipe(RecipeDefinitionName := 'Recipes', RecipeName := 'Automatic');
	recResult := recipieManager.GetRecipeNames('Recipes', ADR(recipeName),1,0);
	recResult := recipieManager.ReadAndSaveRecipe(RecipeDefinitionName := 'Recipes', RecipeName := recipeName);
END_IF

END_FUNCTION

// FBs/Recipie Manangment/SaveValuesPeriodic
FUNCTION SaveValuesPeriodic : DWORD
VAR
	recipieManager : Recipe_Management.RecipeManCommands;
	recipeName : STRING;
	recResult : DWORD;
END_VAR

IF HMIData.bagsMade.count <> 0 THEN
	recResult := recipieManager.CreateRecipe(RecipeDefinitionName := 'Recipes', RecipeName := 'Periodic');
	recResult := recipieManager.GetRecipeNames('Recipes', ADR(recipeName),1,0);
	recResult := recipieManager.ReadAndSaveRecipe(RecipeDefinitionName := 'Recipes', RecipeName := 'Periodic');
END_IF

END_FUNCTION

// FBs/Unused/BagDeliveryFB_BothMotors
FUNCTION_BLOCK BagDeliveryFB_BothMotors EXTENDS BaseComponentFB IMPLEMENTS IComponentStatus
VAR_INPUT
    feedBagPB : BOOL;                // Manually Feed bag out
	jogForwardPB : BOOL;
	jogReversePB : BOOL;
    bagsToFeedSetpoint : INT;        // Bags to feed setpoint for testing
    reverseDistanceSetpoint : REAL := -3;  // Distance to reverse
    bagLengthSetpoint : REAL := 23.5;  // Bag length to feed
    accelSetpoint : INT := 600;            // Acceleration Setpoint
    decelSetpoint : INT := 2000;        // Deceleration Setpoint
    reverseVelocitySetpoint : INT := 3;            // Reverse Velocity setoint (IPS)
    feedVelocitySetpoint : INT := 55;            // Bag Feed Velocity setoint (IPS)
    printVelocitySetpoint : UDINT := 6;            // Print speed (IPS)
    sealOffsetSetpoint : REAL := 1.5;            // Seal Offset
    printOffsetSetpoint : REAL := 3;            // Print Offset
    printLengthSetpoint : REAL := 8;                    // Print length
	reverseToPrintHeadSetpoint : REAL := -1.25;
	feedToPhotoeyeSetpoint : REAL := 2.0;
	useLastPrinterDelta : BOOL := TRUE;
	tensionFailONS : FB_ONS;
END_VAR
VAR_OUTPUT
    state : BAG_DELIVERY_STATES;    // Current state of bag delivery component
	reverseFault : FB_Fault(name := 'Reverse Fault');
	noBagOverEye : FB_Fault(name := 'No bag over Photoeye');
	bagTensionFault : FB_Fault(name := 'Bag Tension Fault');
END_VAR
VAR
    delay : TON := (PT := T#100MS);    // Delay for testing
	jogForwardONS: FB_ONS;
	jogReverseONS: FB_ONS;
	delayForReverseFault : Standard.TON;
	autoFeedDelay : TON := (PT := T#200MS);
	sealBarToPrintHeadLength : REAL;
    bagsCurrentlyFed  :INT;            // Bags currently fed for testing
    remainingLength : REAL;            // Remaining bag length after print
	delayForPrintFeed : TIME := T#250MS;
	printerExtraFeedLength : REAL := 0.25;
    //bagFeedMasterMotor : FB_AppliedMotionStepServoTCP();
    //bagFeedMasterMotor : FB_AppliedMotionBagDeliveryMotor();
	bagFeedMasterMotor : FB_AppliedMotionBagDeliveryMotor_1();
	//bagFeedRearMotor : FB_AppliedMotionBagDeliveryMotor_1();
	bagFeedRearMotor : FB_AppliedMotionStepServoEIPBase();
	accelPercent : REAL := 0.1;
	decelPercent : REAL := 0.05;
    _amReverseBag : BOOL;            // Auto Mode - Reverse bag
    _amFeedBagOut : BOOL;            // Auto Mode - Feed new bag out
    _amWaitForPrinter : BOOL;        // Auto Mode - wait for printer
    _amPrinterReady : BOOL;            // Auto Mode - Printer is ready
    _amStartPrint : BOOL;            // Auto Mode - Start Printing
    _amPrinterDone : BOOL;             // Auto Mode - Printer is Done
	_amFeedToEye : BOOL;			  // Auto Mode - Feed Bag to Eye
END_VAR

//    Function Block: BagDeliveryFB
//    Description: This is the state machine for the bag delivery test rig
//    
//    Created by: Ben Hess
//    Created Date: Thursday, April 19, 2018

SUPER^();
tensionFailONS(CLK := iBagTensionFault);

delay();
delayForReverseFault();
autoFeedDelay(IN := _amFeedBagOut);
// This is the master Applied Motion motor
IF useLastPrinterDelta THEN
	IF Globals.lastPrinterDelta >= T#90MS THEN
		delayForPrintFeed := Globals.lastPrinterDelta - T#80MS;
	ELSE
		delayForPrintFeed := T#10MS;
	END_IF
END_IF
bagLengthSetpoint := HMIData.bagLength;
printVelocitySetpoint := HMIData.printSpeed;
sealOffsetSetpoint := HMIData.bagSkirtLength;
printOffsetSetpoint := HMIData.printOffset;
sealBarToPrintHeadLength := ABS(reverseToPrintHeadSetpoint) + 2.25;
printLengthSetpoint := HMIData.printLength;
reverseVelocitySetpoint := TO_INT(HMIData.bagReverseSpeed);
feedVelocitySetpoint := TO_INT(HMIData.bagForwardSpeed);

